LIN {X 0,Y 401.283,Z 772.145,A -85,B 0,C 180,E1 -11232.942,E2 -11232.942} C_VEL
LIN {X 0,Y 400.696,Z 783.943,A -85,B 0,C 180,E1 -11233.572,E2 -11233.572} C_VEL
LIN {X 0,Y 399.899,Z 796.285,A -85,B 0,C 180,E1 -11234.455,E2 -11234.455} C_VEL
LIN {X 0,Y 399.087,Z 807.279,A -85,B 0,C 180,E1 -11235.468,E2 -11235.468} C_VEL
LIN {X 0,Y 398.218,Z 818.113,A -85,B 0,C 180,E1 -11236.737,E2 -11236.737} C_VEL
LIN {X 0,Y 397.557,Z 826.911,A -85,B 0,C 180,E1 -11238.013,E2 -11238.013} C_VEL
LIN {X 0,Y 396.964,Z 834.155,A -85,B 0,C 180,E1 -11239.288,E2 -11239.288} C_VEL
LIN {X 0,Y 396.505,Z 841.253,A -85,B 0,C 180,E1 -11240.822,E2 -11240.822} C_VEL
LIN {X 0,Y 396.158,Z 846.888,A -85,B 0,C 180,E1 -11242.355,E2 -11242.355} C_VEL
LIN {X 0,Y 395.949,Z 851.307,A -85,B 0,C 180,E1 -11243.887,E2 -11243.887} C_VEL
LIN {X 0,Y 395.956,Z 853.636,A -85,B 0,C 180,E1 -11244.909,E2 -11244.909} C_VEL
LIN {X 0,Y 395.868,Z 855.53,A -85,B 0,C 180,E1 -11245.929,E2 -11245.929} C_VEL
LIN {X 0,Y 395.833,Z 856.959,A -85,B 0,C 180,E1 -11246.948,E2 -11246.948} C_VEL
LIN {X 0,Y 395.901,Z 857.969,A -85,B 0,C 180,E1 -11247.966,E2 -11247.966} C_VEL
LIN {X 0,Y 395.887,Z 858.585,A -85,B 0,C 180,E1 -11248.984,E2 -11248.984} C_VEL
LIN {X 0,Y 395.885,Z 858.804,A -85,B 0,C 180,E1 -11250.001,E2 -11250.001} C_VEL
LIN {X 0,Y 395.896,Z 857.963,A -85,B 0,C 180,E1 -11252.035,E2 -11252.035} C_VEL
LIN {X 0,Y 395.821,Z 856.95,A -85,B 0,C 180,E1 -11253.054,E2 -11253.054} C_VEL
LIN {X 0,Y 395.853,Z 855.516,A -85,B 0,C 180,E1 -11254.073,E2 -11254.073} C_VEL
LIN {X 0,Y 395.924,Z 852.533,A -85,B 0,C 180,E1 -11255.603,E2 -11255.603} C_VEL
LIN {X 0,Y 396.099,Z 848.483,A -85,B 0,C 180,E1 -11257.135,E2 -11257.135} C_VEL
LIN {X 0,Y 396.393,Z 842.229,A -85,B 0,C 180,E1 -11258.925,E2 -11258.925} C_VEL
LIN {X 0,Y 396.861,Z 835.406,A -85,B 0,C 180,E1 -11260.459,E2 -11260.459} C_VEL
LIN {X 0,Y 397.367,Z 828.432,A -85,B 0,C 180,E1 -11261.736,E2 -11261.736} C_VEL
LIN {X 0,Y 398.071,Z 820.005,A -85,B 0,C 180,E1 -11263.01,E2 -11263.01} C_VEL
LIN {X 0,Y 398.827,Z 809.551,A -85,B 0,C 180,E1 -11264.283,E2 -11264.283} C_VEL
LIN {X 0,Y 399.635,Z 799.186,A -85,B 0,C 180,E1 -11265.296,E2 -11265.296} C_VEL
LIN {X 0,Y 400.447,Z 787.762,A -85,B 0,C 180,E1 -11266.178,E2 -11266.178} C_VEL
LIN {X 0,Y 401.084,Z 775.888,A -85,B 0,C 180,E1 -11266.872,E2 -11266.872} C_VEL
LIN {X 0,Y 401.698,Z 763.05,A -85,B 0,C 180,E1 -11267.402,E2 -11267.402} C_VEL
LIN {X 0,Y 402.025,Z 751.019,A -85,B 0,C 180,E1 -11267.716,E2 -11267.716} C_VEL
LIN {X 0,Y 403.019,Z 672.877,A -85,B 0,C 180,E1 -11269.101,E2 -11269.101} C_VEL
LIN {X 0,Y 398.802,Z 636.907,A -85,B 0,C 180,E1 -11269.995,E2 -11269.995} C_VEL
LIN {X 0,Y 398.39,Z 632.093,A -85,B 0,C 180,E1 -11270.256,E2 -11270.256} C_VEL
LIN {X 0,Y 399.692,Z 611.54,A -85,B 0,C 180,E1 -11273.855,E2 -11273.855} C_VEL
LIN {X 0,Y 401.212,Z 590.111,A -85,B 0,C 180,E1 -11277.659,E2 -11277.659} C_VEL
LIN {X 0,Y 402.336,Z 576.283,A -85,B 0,C 180,E1 -11280.146,E2 -11280.146} C_VEL
LIN {X 0,Y 401.749,Z 571.846,A -85,B 0,C 180,E1 -11280.998,E2 -11280.998} C_VEL
LIN {X 0,Y 398.495,Z 556.913,A -85,B 0,C 180,E1 -11284.013,E2 -11284.013} C_VEL
LIN {X 0,Y 397.155,Z 551.015,A -85,B 0,C 180,E1 -11285.255,E2 -11285.255} C_VEL
LIN {X 0,Y 397.133,Z 551.019,A -85,B 0,C 180,E1 -11288.862,E2 -11288.862} C_VEL
LIN {X 0,Y 397.07,Z 551.022,A -85,B 0,C 180,E1 -11292.267,E2 -11292.267} C_VEL
LIN {X 0,Y 397.092,Z 551.018,A -85,B 0,C 180,E1 -11295.068,E2 -11295.068} C_VEL
LIN {X 0,Y 397.07,Z 551.014,A -85,B 0,C 180,E1 -11298.021,E2 -11298.021} C_VEL
LIN {X 0,Y 397.133,Z 551.019,A -85,B 0,C 180,E1 -11301.138,E2 -11301.138} C_VEL
LIN {X 0,Y 397.121,Z 551.01,A -85,B 0,C 180,E1 -11304.496,E2 -11304.496} C_VEL
LIN {X 0,Y 397.079,Z 551.013,A -85,B 0,C 180,E1 -11307.928,E2 -11307.928} C_VEL
LIN {X 0,Y 397.124,Z 551.02,A -85,B 0,C 180,E1 -11311.456,E2 -11311.456} C_VEL
LIN {X 0,Y 397.153,Z 551.003,A -85,B 0,C 180,E1 -11314.488,E2 -11314.488} C_VEL
LIN {X 0,Y 397.096,Z 551.018,A -85,B 0,C 180,E1 -11318.181,E2 -11318.181} C_VEL
LIN {X 0,Y 397.163,Z 550.999,A -85,B 0,C 180,E1 -11321.427,E2 -11321.427} C_VEL
LIN {X 0,Y 397.18,Z 551.005,A -85,B 0,C 180,E1 -11324.608,E2 -11324.608} C_VEL
LIN {X 0,Y 397.22,Z 550.997,A -85,B 0,C 180,E1 -11327.742,E2 -11327.742} C_VEL
LIN {X 0,Y 397.253,Z 550.988,A -85,B 0,C 180,E1 -11330.838,E2 -11330.838} C_VEL
LIN {X 0,Y 397.374,Z 550.985,A -85,B 0,C 180,E1 -11333.909,E2 -11333.909} C_VEL
LIN {X 0,Y 397.449,Z 550.962,A -85,B 0,C 180,E1 -11337.973,E2 -11337.973} C_VEL
LIN {X 0,Y 397.579,Z 550.961,A -85,B 0,C 180,E1 -11340,E2 -11340} C_VEL
LIN {X 0,Y 397.376,Z 550.981,A -85,B 0,C 180,E1 -11343.041,E2 -11343.041} C_VEL
LIN {X 0,Y 397.347,Z 550.978,A -85,B 0,C 180,E1 -11346.639,E2 -11346.639} C_VEL
LIN {X 0,Y 397.257,Z 550.999,A -85,B 0,C 180,E1 -11349.162,E2 -11349.162} C_VEL
LIN {X 0,Y 397.22,Z 550.989,A -85,B 0,C 180,E1 -11352.258,E2 -11352.258} C_VEL
LIN {X 0,Y 397.18,Z 551.008,A -85,B 0,C 180,E1 -11355.392,E2 -11355.392} C_VEL
LIN {X 0,Y 397.163,Z 550.998,A -85,B 0,C 180,E1 -11358.574,E2 -11358.574} C_VEL
LIN {X 0,Y 397.098,Z 551.02,A -85,B 0,C 180,E1 -11361.819,E2 -11361.819} C_VEL
LIN {X 0,Y 397.158,Z 551,A -85,B 0,C 180,E1 -11365.132,E2 -11365.132} C_VEL
LIN {X 0,Y 397.163,Z 551.012,A -85,B 0,C 180,E1 -11367.776,E2 -11367.776} C_VEL
LIN {X 0,Y 397.079,Z 551.013,A -85,B 0,C 180,E1 -11370.883,E2 -11370.883} C_VEL
LIN {X 0,Y 397.127,Z 551.013,A -85,B 0,C 180,E1 -11374.493,E2 -11374.493} C_VEL
LIN {X 0,Y 397.104,Z 551.022,A -85,B 0,C 180,E1 -11378.275,E2 -11378.275} C_VEL
LIN {X 0,Y 397.09,Z 551.022,A -85,B 0,C 180,E1 -11380.909,E2 -11380.909} C_VEL
LIN {X 0,Y 397.103,Z 551.014,A -85,B 0,C 180,E1 -11383.649,E2 -11383.649} C_VEL
LIN {X 0,Y 397.103,Z 551.006,A -85,B 0,C 180,E1 -11386.521,E2 -11386.521} C_VEL
LIN {X 0,Y 397.117,Z 551.018,A -85,B 0,C 180,E1 -11390.423,E2 -11390.423} C_VEL
LIN {X 0,Y 397.111,Z 551.021,A -85,B 0,C 180,E1 -11394.265,E2 -11394.265} C_VEL
LIN {X 0,Y 397.118,Z 551.023,A -85,B 0,C 180,E1 -11396.727,E2 -11396.727} C_VEL
LIN {X 0,Y 397.113,Z 551.129,A -85,B 0,C 180,E1 -11398.278,E2 -11398.278} C_VEL
LIN {X 0,Y 400.541,Z 564.762,A -85,B 0,C 180,E1 -11400.771,E2 -11400.771} C_VEL
LIN {X 0,Y 402.877,Z 576.265,A -85,B 0,C 180,E1 -11402.832,E2 -11402.832} C_VEL
LIN {X 0,Y 401.691,Z 596.601,A -85,B 0,C 180,E1 -11406.062,E2 -11406.062} C_VEL
LIN {X 0,Y 400.709,Z 617.149,A -85,B 0,C 180,E1 -11409.196,E2 -11409.196} C_VEL
LIN {X 0,Y 400.492,Z 622.956,A -85,B 0,C 180,E1 -11410.025,E2 -11410.025} C_VEL
LIN {X 0,Y 403.826,Z 644.421,A -85,B 0,C 180,E1 -11410.601,E2 -11410.601} C_VEL
LIN {X 0,Y 402.635,Z 734.616,A -85,B 0,C 180,E1 -11412.246,E2 -11412.246} C_VEL
LIN {X 0,Y 402.175,Z 747.681,A -85,B 0,C 180,E1 -11412.685,E2 -11412.685} C_VEL
LIN {X 0,Y 401.464,Z 760.645,A -85,B 0,C 180,E1 -11413.341,E2 -11413.341} C_VEL
LIN {X 0,Y 400.81,Z 771.721,A -85,B 0,C 180,E1 -11414.098,E2 -11414.098} C_VEL
LIN {X 0,Y 400.019,Z 782.969,A -85,B 0,C 180,E1 -11415.085,E2 -11415.085} C_VEL
LIN {X 0,Y 399.224,Z 793.487,A -85,B 0,C 180,E1 -11416.251,E2 -11416.251} C_VEL
LIN {X 0,Y 398.405,Z 802.783,A -85,B 0,C 180,E1 -11417.52,E2 -11417.52} C_VEL
LIN {X 0,Y 397.579,Z 811.736,A -85,B 0,C 180,E1 -11419.045,E2 -11419.045} C_VEL
LIN {X 0,Y 396.977,Z 818.928,A -85,B 0,C 180,E1 -11420.574,E2 -11420.574} C_VEL
LIN {X 0,Y 396.426,Z 825.533,A -85,B 0,C 180,E1 -11422.358,E2 -11422.358} C_VEL
LIN {X 0,Y 396.207,Z 829.864,A -85,B 0,C 180,E1 -11423.89,E2 -11423.89} C_VEL
LIN {X 0,Y 396.047,Z 832.144,A -85,B 0,C 180,E1 -11424.909,E2 -11424.909} C_VEL
LIN {X 0,Y 395.878,Z 834.005,A -85,B 0,C 180,E1 -11425.927,E2 -11425.927} C_VEL
LIN {X 0,Y 395.834,Z 836.097,A -85,B 0,C 180,E1 -11427.633,E2 -11427.633} C_VEL
LIN {X 0,Y 395.177,Z 836.822,A -85,B 0,C 180,E1 -11428.477,E2 -11428.477} C_VEL
LIN {X 0,Y 392.325,Z 837.458,A -85,B 0,C 180,E1 -11429.856,E2 -11429.856} C_VEL
LIN {X 0,Y 389.897,Z 837.369,A -85,B 0,C 180,E1 -11430.971,E2 -11430.971} C_VEL
LIN {X 0,Y 388.836,Z 836.891,A -85,B 0,C 180,E1 -11431.83,E2 -11431.83} C_VEL
LIN {X 0,Y 388.741,Z 836.644,A -85,B 0,C 180,E1 -11432.12,E2 -11432.12} C_VEL
LIN {X 0,Y 388.803,Z 834.362,A -85,B 0,C 180,E1 -11434.145,E2 -11434.145} C_VEL
LIN {X 0,Y 389.05,Z 831.49,A -85,B 0,C 180,E1 -11435.701,E2 -11435.701} C_VEL
LIN {X 0,Y 389.251,Z 827.592,A -85,B 0,C 180,E1 -11437.26,E2 -11437.26} C_VEL
LIN {X 0,Y 389.646,Z 822.542,A -85,B 0,C 180,E1 -11438.818,E2 -11438.818} C_VEL
LIN {X 0,Y 390.215,Z 816.176,A -85,B 0,C 180,E1 -11440.375,E2 -11440.375} C_VEL
LIN {X 0,Y 390.943,Z 808.254,A -85,B 0,C 180,E1 -11441.93,E2 -11441.93} C_VEL
LIN {X 0,Y 391.766,Z 800.152,A -85,B 0,C 180,E1 -11443.221,E2 -11443.221} C_VEL
LIN {X 0,Y 392.645,Z 790.211,A -85,B 0,C 180,E1 -11444.511,E2 -11444.511} C_VEL
LIN {X 0,Y 393.477,Z 779.041,A -85,B 0,C 180,E1 -11445.672,E2 -11445.672} C_VEL
LIN {X 0,Y 394.295,Z 768.089,A -85,B 0,C 180,E1 -11446.569,E2 -11446.569} C_VEL
LIN {X 0,Y 395.044,Z 755.761,A -85,B 0,C 180,E1 -11447.336,E2 -11447.336} C_VEL
LIN {X 0,Y 395.619,Z 742.937,A -85,B 0,C 180,E1 -11447.91,E2 -11447.91} C_VEL
LIN {X 0,Y 395.955,Z 730.774,A -85,B 0,C 180,E1 -11448.262,E2 -11448.262} C_VEL
LIN {X 0,Y 397.053,Z 646.296,A -85,B 0,C 180,E1 -11449.808,E2 -11449.808} C_VEL
LIN {X 0,Y 393.25,Z 623.873,A -85,B 0,C 180,E1 -11450.444,E2 -11450.444} C_VEL
LIN {X 0,Y 394.002,Z 604.702,A -85,B 0,C 180,E1 -11453.661,E2 -11453.661} C_VEL
LIN {X 0,Y 395.026,Z 588.085,A -85,B 0,C 180,E1 -11456.62,E2 -11456.62} C_VEL
LIN {X 0,Y 395.615,Z 576.878,A -85,B 0,C 180,E1 -11458.661,E2 -11458.661} C_VEL
LIN {X 0,Y 393.396,Z 565.484,A -85,B 0,C 180,E1 -11460.961,E2 -11460.961} C_VEL
LIN {X 0,Y 390.09,Z 551.892,A -85,B 0,C 180,E1 -11463.796,E2 -11463.796} C_VEL
LIN {X 0,Y 390.056,Z 551.895,A -85,B 0,C 180,E1 -11466.482,E2 -11466.482} C_VEL
LIN {X 0,Y 390.068,Z 551.89,A -85,B 0,C 180,E1 -11469.217,E2 -11469.217} C_VEL
LIN {X 0,Y 390.04,Z 551.896,A -85,B 0,C 180,E1 -11472.373,E2 -11472.373} C_VEL
LIN {X 0,Y 390.096,Z 551.892,A -85,B 0,C 180,E1 -11476.105,E2 -11476.105} C_VEL
LIN {X 0,Y 390.103,Z 551.892,A -85,B 0,C 180,E1 -11478.694,E2 -11478.694} C_VEL
LIN {X 0,Y 395.887,Z 568.43,A -85,B 0,C 180,E1 -11479.322,E2 -11479.322} C_VEL
LIN {X 0,Y 394.931,Z 631.63,A -85,B 0,C 180,E1 -11480.636,E2 -11480.636} C_VEL
LIN {X 0,Y 394.843,Z 645.21,A -85,B 0,C 180,E1 -11481.118,E2 -11481.118} C_VEL
LIN {X 0,Y 394.546,Z 657.641,A -85,B 0,C 180,E1 -11481.757,E2 -11481.757} C_VEL
LIN {X 0,Y 394.14,Z 668.866,A -85,B 0,C 180,E1 -11482.519,E2 -11482.519} C_VEL
LIN {X 0,Y 393.561,Z 680.822,A -85,B 0,C 180,E1 -11483.565,E2 -11483.565} C_VEL
LIN {X 0,Y 392.976,Z 691.857,A -85,B 0,C 180,E1 -11484.777,E2 -11484.777} C_VEL
LIN {X 0,Y 392.361,Z 700.866,A -85,B 0,C 180,E1 -11485.997,E2 -11485.997} C_VEL
LIN {X 0,Y 391.817,Z 709.636,A -85,B 0,C 180,E1 -11487.459,E2 -11487.459} C_VEL
LIN {X 0,Y 391.317,Z 716.667,A -85,B 0,C 180,E1 -11488.892,E2 -11488.892} C_VEL
LIN {X 0,Y 390.858,Z 722.55,A -85,B 0,C 180,E1 -11490.365,E2 -11490.365} C_VEL
LIN {X 0,Y 390.579,Z 728.004,A -85,B 0,C 180,E1 -11492.106,E2 -11492.106} C_VEL
LIN {X 0,Y 390.401,Z 730.789,A -85,B 0,C 180,E1 -11493.253,E2 -11493.253} C_VEL
LIN {X 0,Y 390.269,Z 733.041,A -85,B 0,C 180,E1 -11494.393,E2 -11494.393} C_VEL
LIN {X 0,Y 390.164,Z 734.702,A -85,B 0,C 180,E1 -11495.525,E2 -11495.525} C_VEL
LIN {X 0,Y 390.14,Z 735.967,A -85,B 0,C 180,E1 -11496.735,E2 -11496.735} C_VEL
LIN {X 0,Y 390.156,Z 736.561,A -85,B 0,C 180,E1 -11497.773,E2 -11497.773} C_VEL
LIN {X 0,Y 390.276,Z 736.668,A -85,B 0,C 180,E1 -11499.451,E2 -11499.451} C_VEL
LIN {X 0,Y 390.488,Z 735.718,A -85,B 0,C 180,E1 -11501.097,E2 -11501.097} C_VEL
LIN {X 0,Y 390.712,Z 734.208,A -85,B 0,C 180,E1 -11502.424,E2 -11502.424} C_VEL
LIN {X 0,Y 391.068,Z 731.78,A -85,B 0,C 180,E1 -11503.826,E2 -11503.826} C_VEL
LIN {X 0,Y 391.605,Z 727.154,A -85,B 0,C 180,E1 -11505.717,E2 -11505.717} C_VEL
LIN {X 0,Y 392.359,Z 720.839,A -85,B 0,C 180,E1 -11507.588,E2 -11507.588} C_VEL
LIN {X 0,Y 393.097,Z 713.912,A -85,B 0,C 180,E1 -11509.161,E2 -11509.161} C_VEL
LIN {X 0,Y 393.82,Z 706.604,A -85,B 0,C 180,E1 -11510.498,E2 -11510.498} C_VEL
LIN {X 0,Y 394.597,Z 697.843,A -85,B 0,C 180,E1 -11511.808,E2 -11511.808} C_VEL
LIN {X 0,Y 395.31,Z 688.161,A -85,B 0,C 180,E1 -11512.992,E2 -11512.992} C_VEL
LIN {X 0,Y 396.066,Z 677.186,A -85,B 0,C 180,E1 -11514.059,E2 -11514.059} C_VEL
LIN {X 0,Y 396.643,Z 666.019,A -85,B 0,C 180,E1 -11514.917,E2 -11514.917} C_VEL
LIN {X 0,Y 397.041,Z 654.125,A -85,B 0,C 180,E1 -11515.622,E2 -11515.622} C_VEL
LIN {X 0,Y 397.248,Z 640.901,A -85,B 0,C 180,E1 -11516.174,E2 -11516.174} C_VEL
LIN {X 0,Y 397.271,Z 622.782,A -85,B 0,C 180,E1 -11516.637,E2 -11516.637} C_VEL
LIN {X 0,Y 398.42,Z 570.844,A -85,B 0,C 180,E1 -11517.789,E2 -11517.789} C_VEL
LIN {X 0,Y 392.618,Z 557.28,A -85,B 0,C 180,E1 -11518.541,E2 -11518.541} C_VEL
LIN {X 0,Y 390.462,Z 552.491,A -85,B 0,C 180,E1 -11518.824,E2 -11518.824} C_VEL
LIN {X 0,Y 390.358,Z 551.864,A -85,B 0,C 180,E1 -11518.904,E2 -11518.904} C_VEL
LIN {X 0,Y 390.541,Z 551.84,A -85,B 0,C 180,E1 -11520,E2 -11520} C_VEL
LIN {X 0,Y 390.308,Z 551.867,A -85,B 0,C 180,E1 -11523.097,E2 -11523.097} C_VEL
LIN {X 0,Y 390.33,Z 551.864,A -85,B 0,C 180,E1 -11526.202,E2 -11526.202} C_VEL
LIN {X 0,Y 390.304,Z 551.865,A -85,B 0,C 180,E1 -11528.282,E2 -11528.282} C_VEL
LIN {X 0,Y 390.168,Z 551.881,A -85,B 0,C 180,E1 -11532.483,E2 -11532.483} C_VEL
LIN {X 0,Y 390.129,Z 551.881,A -85,B 0,C 180,E1 -11535.677,E2 -11535.677} C_VEL
LIN {X 0,Y 390.095,Z 551.895,A -85,B 0,C 180,E1 -11538.923,E2 -11538.923} C_VEL
LIN {X 0,Y 390.03,Z 551.901,A -85,B 0,C 180,E1 -11542.235,E2 -11542.235} C_VEL
LIN {X 0,Y 390.11,Z 551.889,A -85,B 0,C 180,E1 -11545.744,E2 -11545.744} C_VEL
LIN {X 0,Y 390.057,Z 551.898,A -85,B 0,C 180,E1 -11549.11,E2 -11549.11} C_VEL
LIN {X 0,Y 390.035,Z 551.902,A -85,B 0,C 180,E1 -11552.722,E2 -11552.722} C_VEL
LIN {X 0,Y 390.05,Z 551.898,A -85,B 0,C 180,E1 -11555.827,E2 -11555.827} C_VEL
LIN {X 0,Y 390.068,Z 551.897,A -85,B 0,C 180,E1 -11559.22,E2 -11559.22} C_VEL
LIN {X 0,Y 390.115,Z 551.891,A -85,B 0,C 180,E1 -11562.388,E2 -11562.388} C_VEL
LIN {X 0,Y 390.113,Z 551.891,A -85,B 0,C 180,E1 -11565.366,E2 -11565.366} C_VEL
LIN {X 0,Y 390.1,Z 551.894,A -85,B 0,C 180,E1 -11568.198,E2 -11568.198} C_VEL
LIN {X 0,Y 390.091,Z 551.895,A -85,B 0,C 180,E1 -11570.91,E2 -11570.91} C_VEL
LIN {X 0,Y 390.083,Z 551.899,A -85,B 0,C 180,E1 -11574.795,E2 -11574.795} C_VEL
LIN {X 0,Y 390.071,Z 551.916,A -85,B 0,C 180,E1 -11575.257,E2 -11575.257} C_VEL
LIN {X 0,Y 393.489,Z 565.056,A -85,B 0,C 180,E1 -11578.207,E2 -11578.207} C_VEL
LIN {X 0,Y 395.857,Z 576.032,A -85,B 0,C 180,E1 -11580.452,E2 -11580.452} C_VEL
LIN {X 0,Y 395.962,Z 579.686,A -85,B 0,C 180,E1 -11581.125,E2 -11581.125} C_VEL
LIN {X 0,Y 393.96,Z 600.394,A -85,B 0,C 180,E1 -11584.652,E2 -11584.652} C_VEL
LIN {X 0,Y 392.222,Z 623.137,A -85,B 0,C 180,E1 -11588.416,E2 -11588.416} C_VEL
LIN {X 0,Y 392.038,Z 625.864,A -85,B 0,C 180,E1 -11588.86,E2 -11588.86} C_VEL
LIN {X 0,Y 394.805,Z 646.803,A -85,B 0,C 180,E1 -11589.542,E2 -11589.542} C_VEL
LIN {X 0,Y 397.038,Z 672.475,A -85,B 0,C 180,E1 -11590.277,E2 -11590.277} C_VEL
LIN {X 0,Y 395.548,Z 739.472,A -85,B 0,C 180,E1 -11591.718,E2 -11591.718} C_VEL
LIN {X 0,Y 395.013,Z 761.303,A -85,B 0,C 180,E1 -11592.229,E2 -11592.229} C_VEL
LIN {X 0,Y 394.404,Z 774.608,A -85,B 0,C 180,E1 -11592.769,E2 -11592.769} C_VEL
LIN {X 0,Y 393.761,Z 785.751,A -85,B 0,C 180,E1 -11593.408,E2 -11593.408} C_VEL
LIN {X 0,Y 392.931,Z 797.671,A -85,B 0,C 180,E1 -11594.305,E2 -11594.305} C_VEL
LIN {X 0,Y 392.079,Z 808.27,A -85,B 0,C 180,E1 -11595.335,E2 -11595.335} C_VEL
LIN {X 0,Y 391.262,Z 817.929,A -85,B 0,C 180,E1 -11596.497,E2 -11596.497} C_VEL
LIN {X 0,Y 390.596,Z 826.726,A -85,B 0,C 180,E1 -11597.796,E2 -11597.796} C_VEL
LIN {X 0,Y 389.95,Z 833.967,A -85,B 0,C 180,E1 -11599.093,E2 -11599.093} C_VEL
LIN {X 0,Y 389.434,Z 841.062,A -85,B 0,C 180,E1 -11600.654,E2 -11600.654} C_VEL
LIN {X 0,Y 389.088,Z 846.697,A -85,B 0,C 180,E1 -11602.215,E2 -11602.215} C_VEL
LIN {X 0,Y 388.836,Z 851.863,A -85,B 0,C 180,E1 -11604.088,E2 -11604.088} C_VEL
LIN {X 0,Y 388.79,Z 855.338,A -85,B 0,C 180,E1 -11605.854,E2 -11605.854} C_VEL
LIN {X 0,Y 388.735,Z 856.767,A -85,B 0,C 180,E1 -11606.892,E2 -11606.892} C_VEL
LIN {X 0,Y 388.798,Z 857.776,A -85,B 0,C 180,E1 -11607.929,E2 -11607.929} C_VEL
LIN {X 0,Y 388.813,Z 858.393,A -85,B 0,C 180,E1 -11608.965,E2 -11608.965} C_VEL
LIN {X 0,Y 388.809,Z 858.612,A -85,B 0,C 180,E1 -11610.001,E2 -11610.001} C_VEL
LIN {X 0,Y 388.786,Z 858.388,A -85,B 0,C 180,E1 -11611.037,E2 -11611.037} C_VEL
LIN {X 0,Y 388.792,Z 857.77,A -85,B 0,C 180,E1 -11612.073,E2 -11612.073} C_VEL
LIN {X 0,Y 388.723,Z 856.757,A -85,B 0,C 180,E1 -11613.11,E2 -11613.11} C_VEL
LIN {X 0,Y 388.776,Z 855.323,A -85,B 0,C 180,E1 -11614.147,E2 -11614.147} C_VEL
LIN {X 0,Y 388.837,Z 851.846,A -85,B 0,C 180,E1 -11615.912,E2 -11615.912} C_VEL
LIN {X 0,Y 389.087,Z 846.672,A -85,B 0,C 180,E1 -11617.787,E2 -11617.787} C_VEL
LIN {X 0,Y 389.491,Z 839.928,A -85,B 0,C 180,E1 -11619.609,E2 -11619.609} C_VEL
LIN {X 0,Y 389.997,Z 832.563,A -85,B 0,C 180,E1 -11621.171,E2 -11621.171} C_VEL
LIN {X 0,Y 390.683,Z 825.051,A -85,B 0,C 180,E1 -11622.467,E2 -11622.467} C_VEL
LIN {X 0,Y 391.366,Z 816.46,A -85,B 0,C 180,E1 -11623.693,E2 -11623.693} C_VEL
LIN {X 0,Y 392.219,Z 805.746,A -85,B 0,C 180,E1 -11624.927,E2 -11624.927} C_VEL
LIN {X 0,Y 393.11,Z 794.436,A -85,B 0,C 180,E1 -11625.955,E2 -11625.955} C_VEL
LIN {X 0,Y 393.998,Z 782.649,A -85,B 0,C 180,E1 -11626.784,E2 -11626.784} C_VEL
LIN {X 0,Y 394.583,Z 770.308,A -85,B 0,C 180,E1 -11627.425,E2 -11627.425} C_VEL
LIN {X 0,Y 395.149,Z 756.569,A -85,B 0,C 180,E1 -11627.901,E2 -11627.901} C_VEL
LIN {X 0,Y 396.063,Z 693.26,A -85,B 0,C 180,E1 -11629.067,E2 -11629.067} C_VEL
LIN {X 0,Y 396.27,Z 673.243,A -85,B 0,C 180,E1 -11629.431,E2 -11629.431} C_VEL
LIN {X 0,Y 391.994,Z 637.185,A -85,B 0,C 180,E1 -11630.338,E2 -11630.338} C_VEL
LIN {X 0,Y 391.513,Z 630.548,A -85,B 0,C 180,E1 -11630.696,E2 -11630.696} C_VEL
LIN {X 0,Y 392.79,Z 610.387,A -85,B 0,C 180,E1 -11634.301,E2 -11634.301} C_VEL
LIN {X 0,Y 394.438,Z 588.982,A -85,B 0,C 180,E1 -11638.176,E2 -11638.176} C_VEL
LIN {X 0,Y 395.386,Z 576.632,A -85,B 0,C 180,E1 -11640.437,E2 -11640.437} C_VEL
LIN {X 0,Y 392.611,Z 563.044,A -85,B 0,C 180,E1 -11643.195,E2 -11643.195} C_VEL
LIN {X 0,Y 390.076,Z 551.897,A -85,B 0,C 180,E1 -11645.598,E2 -11645.598} C_VEL
LIN {X 0,Y 390.073,Z 551.898,A -85,B 0,C 180,E1 -11649.219,E2 -11649.219} C_VEL
LIN {X 0,Y 390.044,Z 551.898,A -85,B 0,C 180,E1 -11652.374,E2 -11652.374} C_VEL
LIN {X 0,Y 390.049,Z 551.899,A -85,B 0,C 180,E1 -11655.355,E2 -11655.355} C_VEL
LIN {X 0,Y 390.034,Z 551.89,A -85,B 0,C 180,E1 -11658.187,E2 -11658.187} C_VEL
LIN {X 0,Y 390.092,Z 551.894,A -85,B 0,C 180,E1 -11660.908,E2 -11660.908} C_VEL
LIN {X 0,Y 390.087,Z 551.888,A -85,B 0,C 180,E1 -11664.793,E2 -11664.793} C_VEL
LIN {X 0,Y 390.024,Z 551.891,A -85,B 0,C 180,E1 -11668.496,E2 -11668.496} C_VEL
LIN {X 0,Y 390.118,Z 551.888,A -85,B 0,C 180,E1 -11672.07,E2 -11672.07} C_VEL
LIN {X 0,Y 390.078,Z 551.882,A -85,B 0,C 180,E1 -11675.519,E2 -11675.519} C_VEL
LIN {X 0,Y 390.056,Z 551.897,A -85,B 0,C 180,E1 -11678.878,E2 -11678.878} C_VEL
LIN {X 0,Y 390.129,Z 551.87,A -85,B 0,C 180,E1 -11682.167,E2 -11682.167} C_VEL
LIN {X 0,Y 390.145,Z 551.887,A -85,B 0,C 180,E1 -11685.393,E2 -11685.393} C_VEL
LIN {X 0,Y 390.148,Z 551.873,A -85,B 0,C 180,E1 -11688.571,E2 -11688.571} C_VEL
LIN {X 0,Y 390.308,Z 551.865,A -85,B 0,C 180,E1 -11692.032,E2 -11692.032} C_VEL
LIN {X 0,Y 390.227,Z 551.872,A -85,B 0,C 180,E1 -11694.834,E2 -11694.834} C_VEL
LIN {X 0,Y 390.418,Z 551.837,A -85,B 0,C 180,E1 -11697.937,E2 -11697.937} C_VEL
LIN {X 0,Y 390.548,Z 551.837,A -85,B 0,C 180,E1 -11700,E2 -11700} C_VEL
LIN {X 0,Y 390.311,Z 551.861,A -85,B 0,C 180,E1 -11703.097,E2 -11703.097} C_VEL
LIN {X 0,Y 390.302,Z 551.856,A -85,B 0,C 180,E1 -11706.634,E2 -11706.634} C_VEL
LIN {X 0,Y 390.209,Z 551.878,A -85,B 0,C 180,E1 -11709.329,E2 -11709.329} C_VEL
LIN {X 0,Y 390.195,Z 551.866,A -85,B 0,C 180,E1 -11713.439,E2 -11713.439} C_VEL
LIN {X 0,Y 390.15,Z 551.883,A -85,B 0,C 180,E1 -11717.308,E2 -11717.308} C_VEL
LIN {X 0,Y 390.088,Z 551.889,A -85,B 0,C 180,E1 -11720.47,E2 -11720.47} C_VEL
LIN {X 0,Y 390.091,Z 551.892,A -85,B 0,C 180,E1 -11723.351,E2 -11723.351} C_VEL
LIN {X 0,Y 390.115,Z 551.886,A -85,B 0,C 180,E1 -11726.768,E2 -11726.768} C_VEL
LIN {X 0,Y 390.04,Z 551.891,A -85,B 0,C 180,E1 -11730.3,E2 -11730.3} C_VEL
LIN {X 0,Y 390.07,Z 551.898,A -85,B 0,C 180,E1 -11734.025,E2 -11734.025} C_VEL
LIN {X 0,Y 390.045,Z 551.9,A -85,B 0,C 180,E1 -11737.551,E2 -11737.551} C_VEL
LIN {X 0,Y 390.058,Z 551.898,A -85,B 0,C 180,E1 -11740.821,E2 -11740.821} C_VEL
LIN {X 0,Y 390.056,Z 551.893,A -85,B 0,C 180,E1 -11743.886,E2 -11743.886} C_VEL
LIN {X 0,Y 390.058,Z 551.881,A -85,B 0,C 180,E1 -11746.789,E2 -11746.789} C_VEL
LIN {X 0,Y 390.058,Z 551.897,A -85,B 0,C 180,E1 -11749.56,E2 -11749.56} C_VEL
LIN {X 0,Y 390.047,Z 551.89,A -85,B 0,C 180,E1 -11752.449,E2 -11752.449} C_VEL
LIN {X 0,Y 390.071,Z 551.898,A -85,B 0,C 180,E1 -11755.975,E2 -11755.975} C_VEL
LIN {X 0,Y 390.045,Z 551.911,A -85,B 0,C 180,E1 -11757.873,E2 -11757.873} C_VEL
LIN {X 0,Y 393.337,Z 564.739,A -85,B 0,C 180,E1 -11760.251,E2 -11760.251} C_VEL
LIN {X 0,Y 396.036,Z 577.286,A -85,B 0,C 180,E1 -11762.536,E2 -11762.536} C_VEL
LIN {X 0,Y 395.514,Z 587.469,A -85,B 0,C 180,E1 -11764.192,E2 -11764.192} C_VEL
LIN {X 0,Y 394.21,Z 610.213,A -85,B 0,C 180,E1 -11767.765,E2 -11767.765} C_VEL
LIN {X 0,Y 393.698,Z 623.087,A -85,B 0,C 180,E1 -11769.665,E2 -11769.665} C_VEL
LIN {X 0,Y 397.139,Z 644.951,A -85,B 0,C 180,E1 -11770.269,E2 -11770.269} C_VEL
LIN {X 0,Y 395.903,Z 734.743,A -85,B 0,C 180,E1 -11771.934,E2 -11771.934} C_VEL
LIN {X 0,Y 395.419,Z 747.843,A -85,B 0,C 180,E1 -11772.379,E2 -11772.379} C_VEL
LIN {X 0,Y 394.672,Z 760.818,A -85,B 0,C 180,E1 -11773.046,E2 -11773.046} C_VEL
LIN {X 0,Y 394.001,Z 771.9,A -85,B 0,C 180,E1 -11773.816,E2 -11773.816} C_VEL
LIN {X 0,Y 393.174,Z 783.072,A -85,B 0,C 180,E1 -11774.811,E2 -11774.811} C_VEL
LIN {X 0,Y 392.35,Z 793.674,A -85,B 0,C 180,E1 -11776.005,E2 -11776.005} C_VEL
LIN {X 0,Y 391.469,Z 802.973,A -85,B 0,C 180,E1 -11777.295,E2 -11777.295} C_VEL
LIN {X 0,Y 390.621,Z 811.927,A -85,B 0,C 180,E1 -11778.847,E2 -11778.847} C_VEL
LIN {X 0,Y 389.958,Z 819.12,A -85,B 0,C 180,E1 -11780.403,E2 -11780.403} C_VEL
LIN {X 0,Y 389.373,Z 825.726,A -85,B 0,C 180,E1 -11782.219,E2 -11782.219} C_VEL
LIN {X 0,Y 389.132,Z 830.057,A -85,B 0,C 180,E1 -11783.778,E2 -11783.778} C_VEL
LIN {X 0,Y 388.993,Z 832.337,A -85,B 0,C 180,E1 -11784.816,E2 -11784.816} C_VEL
LIN {X 0,Y 388.805,Z 834.198,A -85,B 0,C 180,E1 -11785.853,E2 -11785.853} C_VEL
LIN {X 0,Y 388.738,Z 836.329,A -85,B 0,C 180,E1 -11787.63,E2 -11787.63} C_VEL
LIN {X 0,Y 388.728,Z 837.229,A -85,B 0,C 180,E1 -11788.963,E2 -11788.963} C_VEL
LIN {X 0,Y 388.708,Z 837.465,A -85,B 0,C 180,E1 -11789.999,E2 -11789.999} C_VEL
LIN {X 0,Y 388.728,Z 837.274,A -85,B 0,C 180,E1 -11791.035,E2 -11791.035} C_VEL
LIN {X 0,Y 388.741,Z 836.644,A -85,B 0,C 180,E1 -11792.12,E2 -11792.12} C_VEL
LIN {X 0,Y 388.058,Z 835.905,A -85,B 0,C 180,E1 -11792.976,E2 -11792.976} C_VEL
LIN {X 0,Y 385.262,Z 834.163,A -85,B 0,C 180,E1 -11794.363,E2 -11794.363} C_VEL
LIN {X 0,Y 382.985,Z 832.294,A -85,B 0,C 180,E1 -11795.468,E2 -11795.468} C_VEL
LIN {X 0,Y 382.107,Z 830.538,A -85,B 0,C 180,E1 -11796.308,E2 -11796.308} C_VEL
LIN {X 0,Y 382.087,Z 829.881,A -85,B 0,C 180,E1 -11796.589,E2 -11796.589} C_VEL
LIN {X 0,Y 382.461,Z 824.529,A -85,B 0,C 180,E1 -11798.452,E2 -11798.452} C_VEL
LIN {X 0,Y 383.029,Z 818.635,A -85,B 0,C 180,E1 -11800.037,E2 -11800.037} C_VEL
LIN {X 0,Y 383.718,Z 811.296,A -85,B 0,C 180,E1 -11801.622,E2 -11801.622} C_VEL
LIN {X 0,Y 384.461,Z 803.784,A -85,B 0,C 180,E1 -11802.939,E2 -11802.939} C_VEL
LIN {X 0,Y 385.51,Z 793.585,A -85,B 0,C 180,E1 -11804.381,E2 -11804.381} C_VEL
LIN {X 0,Y 386.36,Z 782.728,A -85,B 0,C 180,E1 -11805.619,E2 -11805.619} C_VEL
LIN {X 0,Y 387.258,Z 771.636,A -85,B 0,C 180,E1 -11806.607,E2 -11806.607} C_VEL
LIN {X 0,Y 388.098,Z 759.358,A -85,B 0,C 180,E1 -11807.452,E2 -11807.452} C_VEL
LIN {X 0,Y 388.733,Z 746.404,A -85,B 0,C 180,E1 -11808.102,E2 -11808.102} C_VEL
LIN {X 0,Y 389.174,Z 733.502,A -85,B 0,C 180,E1 -11808.524,E2 -11808.524} C_VEL
LIN {X 0,Y 390.406,Z 647.315,A -85,B 0,C 180,E1 -11810.141,E2 -11810.141} C_VEL
LIN {X 0,Y 386.419,Z 623.901,A -85,B 0,C 180,E1 -11810.844,E2 -11810.844} C_VEL
LIN {X 0,Y 387.181,Z 606.286,A -85,B 0,C 180,E1 -11813.819,E2 -11813.819} C_VEL
LIN {X 0,Y 388.251,Z 589.054,A -85,B 0,C 180,E1 -11816.905,E2 -11816.905} C_VEL
LIN {X 0,Y 388.776,Z 578.115,A -85,B 0,C 180,E1 -11818.917,E2 -11818.917} C_VEL
LIN {X 0,Y 386.222,Z 565.725,A -85,B 0,C 180,E1 -11821.458,E2 -11821.458} C_VEL
LIN {X 0,Y 383.013,Z 552.776,A -85,B 0,C 180,E1 -11824.191,E2 -11824.191} C_VEL
LIN {X 0,Y 382.994,Z 552.782,A -85,B 0,C 180,E1 -11827.267,E2 -11827.267} C_VEL
LIN {X 0,Y 383.005,Z 552.77,A -85,B 0,C 180,E1 -11829.957,E2 -11829.957} C_VEL
LIN {X 0,Y 383,Z 552.766,A -85,B 0,C 180,E1 -11832.777,E2 -11832.777} C_VEL
LIN {X 0,Y 383.033,Z 552.773,A -85,B 0,C 180,E1 -11835.794,E2 -11835.794} C_VEL
LIN {X 0,Y 383.081,Z 552.767,A -85,B 0,C 180,E1 -11838.387,E2 -11838.387} C_VEL
LIN {X 0,Y 389.013,Z 569.772,A -85,B 0,C 180,E1 -11839.055,E2 -11839.055} C_VEL
LIN {X 0,Y 388.083,Z 632.568,A -85,B 0,C 180,E1 -11840.393,E2 -11840.393} C_VEL
LIN {X 0,Y 387.971,Z 646.052,A -85,B 0,C 180,E1 -11840.88,E2 -11840.88} C_VEL
LIN {X 0,Y 387.656,Z 658.819,A -85,B 0,C 180,E1 -11841.549,E2 -11841.549} C_VEL
LIN {X 0,Y 387.181,Z 671.323,A -85,B 0,C 180,E1 -11842.434,E2 -11842.434} C_VEL
LIN {X 0,Y 386.625,Z 682.659,A -85,B 0,C 180,E1 -11843.464,E2 -11843.464} C_VEL
LIN {X 0,Y 386.051,Z 692.741,A -85,B 0,C 180,E1 -11844.598,E2 -11844.598} C_VEL
LIN {X 0,Y 385.394,Z 702.11,A -85,B 0,C 180,E1 -11845.892,E2 -11845.892} C_VEL
LIN {X 0,Y 384.78,Z 711.29,A -85,B 0,C 180,E1 -11847.461,E2 -11847.461} C_VEL
LIN {X 0,Y 384.291,Z 718.091,A -85,B 0,C 180,E1 -11848.892,E2 -11848.892} C_VEL
LIN {X 0,Y 383.824,Z 723.831,A -85,B 0,C 180,E1 -11850.371,E2 -11850.371} C_VEL
LIN {X 0,Y 383.555,Z 729.21,A -85,B 0,C 180,E1 -11852.144,E2 -11852.144} C_VEL
LIN {X 0,Y 383.29,Z 733.253,A -85,B 0,C 180,E1 -11853.953,E2 -11853.953} C_VEL
LIN {X 0,Y 383.184,Z 735.08,A -85,B 0,C 180,E1 -11855.049,E2 -11855.049} C_VEL
LIN {X 0,Y 383.106,Z 736.769,A -85,B 0,C 180,E1 -11856.522,E2 -11856.522} C_VEL
LIN {X 0,Y 383.173,Z 737.797,A -85,B 0,C 180,E1 -11858.48,E2 -11858.48} C_VEL
LIN {X 0,Y 383.278,Z 737.701,A -85,B 0,C 180,E1 -11859.611,E2 -11859.611} C_VEL
LIN {X 0,Y 383.434,Z 737.167,A -85,B 0,C 180,E1 -11860.736,E2 -11860.736} C_VEL
LIN {X 0,Y 383.671,Z 735.655,A -85,B 0,C 180,E1 -11862.268,E2 -11862.268} C_VEL
LIN {X 0,Y 384.145,Z 732.706,A -85,B 0,C 180,E1 -11864.072,E2 -11864.072} C_VEL
LIN {X 0,Y 384.598,Z 729.182,A -85,B 0,C 180,E1 -11865.574,E2 -11865.574} C_VEL
LIN {X 0,Y 385.307,Z 723.609,A -85,B 0,C 180,E1 -11867.357,E2 -11867.357} C_VEL
LIN {X 0,Y 386.116,Z 716.774,A -85,B 0,C 180,E1 -11869.035,E2 -11869.035} C_VEL
LIN {X 0,Y 386.981,Z 708.801,A -85,B 0,C 180,E1 -11870.593,E2 -11870.593} C_VEL
LIN {X 0,Y 387.772,Z 700.306,A -85,B 0,C 180,E1 -11871.925,E2 -11871.925} C_VEL
LIN {X 0,Y 388.556,Z 690.663,A -85,B 0,C 180,E1 -11873.157,E2 -11873.157} C_VEL
LIN {X 0,Y 389.362,Z 679.833,A -85,B 0,C 180,E1 -11874.268,E2 -11874.268} C_VEL
LIN {X 0,Y 390.037,Z 667.89,A -85,B 0,C 180,E1 -11875.22,E2 -11875.22} C_VEL
LIN {X 0,Y 390.509,Z 654.994,A -85,B 0,C 180,E1 -11876.001,E2 -11876.001} C_VEL
LIN {X 0,Y 390.731,Z 641.923,A -85,B 0,C 180,E1 -11876.552,E2 -11876.552} C_VEL
LIN {X 0,Y 390.772,Z 623.164,A -85,B 0,C 180,E1 -11877.043,E2 -11877.043} C_VEL
LIN {X 0,Y 392.006,Z 572.731,A -85,B 0,C 180,E1 -11878.192,E2 -11878.192} C_VEL
LIN {X 0,Y 386.596,Z 560.133,A -85,B 0,C 180,E1 -11878.92,E2 -11878.92} C_VEL
LIN {X 0,Y 383.49,Z 553.413,A -85,B 0,C 180,E1 -11879.344,E2 -11879.344} C_VEL
LIN {X 0,Y 383.375,Z 552.734,A -85,B 0,C 180,E1 -11879.409,E2 -11879.409} C_VEL
LIN {X 0,Y 383.314,Z 552.741,A -85,B 0,C 180,E1 -11881.051,E2 -11881.051} C_VEL
LIN {X 0,Y 383.245,Z 552.747,A -85,B 0,C 180,E1 -11883.154,E2 -11883.154} C_VEL
LIN {X 0,Y 383.286,Z 552.742,A -85,B 0,C 180,E1 -11886.316,E2 -11886.316} C_VEL
LIN {X 0,Y 383.25,Z 552.745,A -85,B 0,C 180,E1 -11888.436,E2 -11888.436} C_VEL
LIN {X 0,Y 383.097,Z 552.764,A -85,B 0,C 180,E1 -11891.642,E2 -11891.642} C_VEL
LIN {X 0,Y 383.102,Z 552.762,A -85,B 0,C 180,E1 -11894.882,E2 -11894.882} C_VEL
LIN {X 0,Y 383.079,Z 552.766,A -85,B 0,C 180,E1 -11898.173,E2 -11898.173} C_VEL
LIN {X 0,Y 382.983,Z 552.778,A -85,B 0,C 180,E1 -11901.532,E2 -11901.532} C_VEL
LIN {X 0,Y 383.043,Z 552.773,A -85,B 0,C 180,E1 -11904.961,E2 -11904.961} C_VEL
LIN {X 0,Y 383.04,Z 552.772,A -85,B 0,C 180,E1 -11908.493,E2 -11908.493} C_VEL
LIN {X 0,Y 383.003,Z 552.776,A -85,B 0,C 180,E1 -11912.15,E2 -11912.15} C_VEL
LIN {X 0,Y 383.01,Z 552.771,A -85,B 0,C 180,E1 -11914.669,E2 -11914.669} C_VEL
LIN {X 0,Y 382.996,Z 552.773,A -85,B 0,C 180,E1 -11917.906,E2 -11917.906} C_VEL
LIN {X 0,Y 383.04,Z 552.775,A -85,B 0,C 180,E1 -11921.34,E2 -11921.34} C_VEL
LIN {X 0,Y 383.063,Z 552.772,A -85,B 0,C 180,E1 -11924.316,E2 -11924.316} C_VEL
LIN {X 0,Y 383.069,Z 552.768,A -85,B 0,C 180,E1 -11927.25,E2 -11927.25} C_VEL
LIN {X 0,Y 383.018,Z 552.775,A -85,B 0,C 180,E1 -11930.413,E2 -11930.413} C_VEL
LIN {X 0,Y 383.023,Z 552.779,A -85,B 0,C 180,E1 -11934.046,E2 -11934.046} C_VEL
LIN {X 0,Y 383.055,Z 552.933,A -85,B 0,C 180,E1 -11934.736,E2 -11934.736} C_VEL
LIN {X 0,Y 385.913,Z 563.614,A -85,B 0,C 180,E1 -11937.254,E2 -11937.254} C_VEL
LIN {X 0,Y 388.69,Z 575.718,A -85,B 0,C 180,E1 -11939.853,E2 -11939.853} C_VEL
LIN {X 0,Y 389.285,Z 579.464,A -85,B 0,C 180,E1 -11940.607,E2 -11940.607} C_VEL
LIN {X 0,Y 387.538,Z 596.64,A -85,B 0,C 180,E1 -11943.622,E2 -11943.622} C_VEL
LIN {X 0,Y 385.709,Z 617.795,A -85,B 0,C 180,E1 -11947.221,E2 -11947.221} C_VEL
LIN {X 0,Y 385.222,Z 624.537,A -85,B 0,C 180,E1 -11948.355,E2 -11948.355} C_VEL
LIN {X 0,Y 388.031,Z 645.109,A -85,B 0,C 180,E1 -11949.064,E2 -11949.064} C_VEL
LIN {X 0,Y 390.138,Z 668.772,A -85,B 0,C 180,E1 -11949.763,E2 -11949.763} C_VEL
LIN {X 0,Y 390.407,Z 676.656,A -85,B 0,C 180,E1 -11949.966,E2 -11949.966} C_VEL
LIN {X 0,Y 388.901,Z 738.029,A -85,B 0,C 180,E1 -11951.326,E2 -11951.326} C_VEL
LIN {X 0,Y 388.645,Z 747.872,A -85,B 0,C 180,E1 -11951.586,E2 -11951.586} C_VEL
LIN {X 0,Y 388.277,Z 761.184,A -85,B 0,C 180,E1 -11951.91,E2 -11951.91} C_VEL
LIN {X 0,Y 387.613,Z 774.457,A -85,B 0,C 180,E1 -11952.457,E2 -11952.457} C_VEL
LIN {X 0,Y 386.807,Z 787.544,A -85,B 0,C 180,E1 -11953.237,E2 -11953.237} C_VEL
LIN {X 0,Y 385.952,Z 798.924,A -85,B 0,C 180,E1 -11954.15,E2 -11954.15} C_VEL
LIN {X 0,Y 385.095,Z 809.257,A -85,B 0,C 180,E1 -11955.198,E2 -11955.198} C_VEL
LIN {X 0,Y 384.211,Z 819.684,A -85,B 0,C 180,E1 -11956.514,E2 -11956.514} C_VEL
LIN {X 0,Y 383.483,Z 828.104,A -85,B 0,C 180,E1 -11957.834,E2 -11957.834} C_VEL
LIN {X 0,Y 382.746,Z 836.303,A -85,B 0,C 180,E1 -11959.42,E2 -11959.42} C_VEL
LIN {X 0,Y 382.283,Z 842.891,A -85,B 0,C 180,E1 -11961.011,E2 -11961.011} C_VEL
LIN {X 0,Y 381.946,Z 848.122,A -85,B 0,C 180,E1 -11962.601,E2 -11962.601} C_VEL
LIN {X 0,Y 381.737,Z 852.045,A -85,B 0,C 180,E1 -11964.137,E2 -11964.137} C_VEL
LIN {X 0,Y 381.714,Z 855.146,A -85,B 0,C 180,E1 -11965.777,E2 -11965.777} C_VEL
LIN {X 0,Y 381.642,Z 856.574,A -85,B 0,C 180,E1 -11966.834,E2 -11966.834} C_VEL
LIN {X 0,Y 381.694,Z 857.583,A -85,B 0,C 180,E1 -11967.891,E2 -11967.891} C_VEL
LIN {X 0,Y 381.741,Z 858.201,A -85,B 0,C 180,E1 -11968.946,E2 -11968.946} C_VEL
LIN {X 0,Y 381.735,Z 858.42,A -85,B 0,C 180,E1 -11970.001,E2 -11970.001} C_VEL
LIN {X 0,Y 381.716,Z 858.196,A -85,B 0,C 180,E1 -11971.056,E2 -11971.056} C_VEL
LIN {X 0,Y 381.688,Z 857.576,A -85,B 0,C 180,E1 -11972.111,E2 -11972.111} C_VEL
LIN {X 0,Y 381.63,Z 856.564,A -85,B 0,C 180,E1 -11973.168,E2 -11973.168} C_VEL
LIN {X 0,Y 381.701,Z 855.13,A -85,B 0,C 180,E1 -11974.224,E2 -11974.224} C_VEL
LIN {X 0,Y 381.737,Z 852.03,A -85,B 0,C 180,E1 -11975.862,E2 -11975.862} C_VEL
LIN {X 0,Y 381.958,Z 848.097,A -85,B 0,C 180,E1 -11977.401,E2 -11977.401} C_VEL
LIN {X 0,Y 382.296,Z 841.843,A -85,B 0,C 180,E1 -11979.257,E2 -11979.257} C_VEL
LIN {X 0,Y 382.795,Z 835.022,A -85,B 0,C 180,E1 -11980.848,E2 -11980.848} C_VEL
LIN {X 0,Y 383.443,Z 828.052,A -85,B 0,C 180,E1 -11982.169,E2 -11982.169} C_VEL
LIN {X 0,Y 384.18,Z 819.628,A -85,B 0,C 180,E1 -11983.489,E2 -11983.489} C_VEL
LIN {X 0,Y 385.043,Z 809.18,A -85,B 0,C 180,E1 -11984.806,E2 -11984.806} C_VEL
LIN {X 0,Y 385.922,Z 798.823,A -85,B 0,C 180,E1 -11985.853,E2 -11985.853} C_VEL
LIN {X 0,Y 386.808,Z 787.411,A -85,B 0,C 180,E1 -11986.765,E2 -11986.765} C_VEL
LIN {X 0,Y 387.495,Z 775.556,A -85,B 0,C 180,E1 -11987.482,E2 -11987.482} C_VEL
LIN {X 0,Y 388.177,Z 762.754,A -85,B 0,C 180,E1 -11988.029,E2 -11988.029} C_VEL
LIN {X 0,Y 388.557,Z 750.806,A -85,B 0,C 180,E1 -11988.351,E2 -11988.351} C_VEL
LIN {X 0,Y 389.553,Z 673.809,A -85,B 0,C 180,E1 -11989.768,E2 -11989.768} C_VEL
LIN {X 0,Y 385.462,Z 638.824,A -85,B 0,C 180,E1 -11990.662,E2 -11990.662} C_VEL
LIN {X 0,Y 384.993,Z 634.332,A -85,B 0,C 180,E1 -11990.863,E2 -11990.863} C_VEL
LIN {X 0,Y 384.587,Z 628.881,A -85,B 0,C 180,E1 -11991.172,E2 -11991.172} C_VEL
LIN {X 0,Y 385.923,Z 609.198,A -85,B 0,C 180,E1 -11994.763,E2 -11994.763} C_VEL
LIN {X 0,Y 387.657,Z 587.77,A -85,B 0,C 180,E1 -11998.714,E2 -11998.714} C_VEL
LIN {X 0,Y 388.457,Z 578.542,A -85,B 0,C 180,E1 -12000.437,E2 -12000.437} C_VEL
LIN {X 0,Y 386.641,Z 568.814,A -85,B 0,C 180,E1 -12002.427,E2 -12002.427} C_VEL
LIN {X 0,Y 383.292,Z 553.909,A -85,B 0,C 180,E1 -12005.603,E2 -12005.603} C_VEL
LIN {X 0,Y 383.012,Z 552.776,A -85,B 0,C 180,E1 -12005.876,E2 -12005.876} C_VEL
LIN {X 0,Y 383.018,Z 552.775,A -85,B 0,C 180,E1 -12009.587,E2 -12009.587} C_VEL
LIN {X 0,Y 383.007,Z 552.778,A -85,B 0,C 180,E1 -12012.779,E2 -12012.779} C_VEL
LIN {X 0,Y 383.002,Z 552.776,A -85,B 0,C 180,E1 -12015.79,E2 -12015.79} C_VEL
LIN {X 0,Y 382.99,Z 552.768,A -85,B 0,C 180,E1 -12018.796,E2 -12018.796} C_VEL
LIN {X 0,Y 383.002,Z 552.771,A -85,B 0,C 180,E1 -12022.096,E2 -12022.096} C_VEL
LIN {X 0,Y 383.02,Z 552.775,A -85,B 0,C 180,E1 -12025.332,E2 -12025.332} C_VEL
LIN {X 0,Y 382.984,Z 552.766,A -85,B 0,C 180,E1 -12029.081,E2 -12029.081} C_VEL
LIN {X 0,Y 383.058,Z 552.768,A -85,B 0,C 180,E1 -12032.698,E2 -12032.698} C_VEL
LIN {X 0,Y 383.051,Z 552.757,A -85,B 0,C 180,E1 -12035.04,E2 -12035.04} C_VEL
LIN {X 0,Y 382.993,Z 552.775,A -85,B 0,C 180,E1 -12038.469,E2 -12038.469} C_VEL
LIN {X 0,Y 383.064,Z 552.75,A -85,B 0,C 180,E1 -12041.826,E2 -12041.826} C_VEL
LIN {X 0,Y 383.111,Z 552.76,A -85,B 0,C 180,E1 -12045.118,E2 -12045.118} C_VEL
LIN {X 0,Y 383.097,Z 552.751,A -85,B 0,C 180,E1 -12048.358,E2 -12048.358} C_VEL
LIN {X 0,Y 383.264,Z 552.743,A -85,B 0,C 180,E1 -12051.976,E2 -12051.976} C_VEL
LIN {X 0,Y 383.199,Z 552.747,A -85,B 0,C 180,E1 -12054.739,E2 -12054.739} C_VEL
LIN {X 0,Y 383.385,Z 552.712,A -85,B 0,C 180,E1 -12057.899,E2 -12057.899} C_VEL
LIN {X 0,Y 383.518,Z 552.713,A -85,B 0,C 180,E1 -12060,E2 -12060} C_VEL
LIN {X 0,Y 383.248,Z 552.741,A -85,B 0,C 180,E1 -12063.154,E2 -12063.154} C_VEL
LIN {X 0,Y 383.262,Z 552.734,A -85,B 0,C 180,E1 -12066.626,E2 -12066.626} C_VEL
LIN {X 0,Y 383.155,Z 552.758,A -85,B 0,C 180,E1 -12069.502,E2 -12069.502} C_VEL
LIN {X 0,Y 383.126,Z 552.747,A -85,B 0,C 180,E1 -12073.536,E2 -12073.536} C_VEL
LIN {X 0,Y 383.096,Z 552.763,A -85,B 0,C 180,E1 -12077.455,E2 -12077.455} C_VEL
LIN {X 0,Y 383.03,Z 552.768,A -85,B 0,C 180,E1 -12080.647,E2 -12080.647} C_VEL
LIN {X 0,Y 383.034,Z 552.769,A -85,B 0,C 180,E1 -12083.807,E2 -12083.807} C_VEL
LIN {X 0,Y 383.081,Z 552.757,A -85,B 0,C 180,E1 -12086.123,E2 -12086.123} C_VEL
LIN {X 0,Y 382.993,Z 552.775,A -85,B 0,C 180,E1 -12089.7,E2 -12089.7} C_VEL
LIN {X 0,Y 383.005,Z 552.776,A -85,B 0,C 180,E1 -12093.401,E2 -12093.401} C_VEL
LIN {X 0,Y 383.033,Z 552.769,A -85,B 0,C 180,E1 -12096.165,E2 -12096.165} C_VEL
LIN {X 0,Y 383.01,Z 552.772,A -85,B 0,C 180,E1 -12099.958,E2 -12099.958} C_VEL
LIN {X 0,Y 383.007,Z 552.77,A -85,B 0,C 180,E1 -12102.779,E2 -12102.779} C_VEL
LIN {X 0,Y 382.999,Z 552.774,A -85,B 0,C 180,E1 -12105.789,E2 -12105.789} C_VEL
LIN {X 0,Y 382.989,Z 552.772,A -85,B 0,C 180,E1 -12108.796,E2 -12108.796} C_VEL
LIN {X 0,Y 383.003,Z 552.765,A -85,B 0,C 180,E1 -12112.096,E2 -12112.096} C_VEL
LIN {X 0,Y 383.021,Z 552.776,A -85,B 0,C 180,E1 -12115.332,E2 -12115.332} C_VEL
LIN {X 0,Y 383.034,Z 552.955,A -85,B 0,C 180,E1 -12117.474,E2 -12117.474} C_VEL
LIN {X 0,Y 386.479,Z 566.231,A -85,B 0,C 180,E1 -12119.995,E2 -12119.995} C_VEL
LIN {X 0,Y 389.131,Z 578.45,A -85,B 0,C 180,E1 -12122.249,E2 -12122.249} C_VEL
LIN {X 0,Y 389.175,Z 582.468,A -85,B 0,C 180,E1 -12122.931,E2 -12122.931} C_VEL
LIN {X 0,Y 387.809,Z 603.008,A -85,B 0,C 180,E1 -12126.22,E2 -12126.22} C_VEL
LIN {X 0,Y 387.018,Z 621.241,A -85,B 0,C 180,E1 -12129.01,E2 -12129.01} C_VEL
LIN {X 0,Y 386.989,Z 623.532,A -85,B 0,C 180,E1 -12129.308,E2 -12129.308} C_VEL
LIN {X 0,Y 390.474,Z 645.902,A -85,B 0,C 180,E1 -12129.934,E2 -12129.934} C_VEL
LIN {X 0,Y 389.169,Z 734.871,A -85,B 0,C 180,E1 -12131.61,E2 -12131.61} C_VEL
LIN {X 0,Y 388.67,Z 748.004,A -85,B 0,C 180,E1 -12132.063,E2 -12132.063} C_VEL
LIN {X 0,Y 387.893,Z 760.991,A -85,B 0,C 180,E1 -12132.741,E2 -12132.741} C_VEL
LIN {X 0,Y 387.208,Z 772.08,A -85,B 0,C 180,E1 -12133.524,E2 -12133.524} C_VEL
LIN {X 0,Y 386.409,Z 782.183,A -85,B 0,C 180,E1 -12134.425,E2 -12134.425} C_VEL
LIN {X 0,Y 385.58,Z 792.826,A -85,B 0,C 180,E1 -12135.62,E2 -12135.62} C_VEL
LIN {X 0,Y 384.547,Z 803.162,A -85,B 0,C 180,E1 -12137.062,E2 -12137.062} C_VEL
LIN {X 0,Y 383.797,Z 810.785,A -85,B 0,C 180,E1 -12138.379,E2 -12138.379} C_VEL
LIN {X 0,Y 383.08,Z 818.223,A -85,B 0,C 180,E1 -12139.962,E2 -12139.962} C_VEL
LIN {X 0,Y 382.471,Z 824.198,A -85,B 0,C 180,E1 -12141.546,E2 -12141.546} C_VEL
LIN {X 0,Y 382.16,Z 829.232,A -85,B 0,C 180,E1 -12143.254,E2 -12143.254} C_VEL
LIN {X 0,Y 381.918,Z 832.53,A -85,B 0,C 180,E1 -12144.72,E2 -12144.72} C_VEL
LIN {X 0,Y 381.736,Z 834.391,A -85,B 0,C 180,E1 -12145.776,E2 -12145.776} C_VEL
LIN {X 0,Y 381.667,Z 835.813,A -85,B 0,C 180,E1 -12146.832,E2 -12146.832} C_VEL
LIN {X 0,Y 381.643,Z 837.422,A -85,B 0,C 180,E1 -12148.944,E2 -12148.944} C_VEL
LIN {X 0,Y 381.64,Z 837.657,A -85,B 0,C 180,E1 -12149.999,E2 -12149.999} C_VEL
LIN {X 0,Y 381.643,Z 837.466,A -85,B 0,C 180,E1 -12151.054,E2 -12151.054} C_VEL
LIN {X 0,Y 381.655,Z 835.917,A -85,B 0,C 180,E1 -12153.166,E2 -12153.166} C_VEL
LIN {X 0,Y 381.734,Z 834.553,A -85,B 0,C 180,E1 -12154.222,E2 -12154.222} C_VEL
LIN {X 0,Y 381.986,Z 831.681,A -85,B 0,C 180,E1 -12155.807,E2 -12155.807} C_VEL
LIN {X 0,Y 382.087,Z 829.881,A -85,B 0,C 180,E1 -12156.589,E2 -12156.589} C_VEL
LIN {X 0,Y 381.613,Z 827.821,A -85,B 0,C 180,E1 -12157.416,E2 -12157.416} C_VEL
LIN {X 0,Y 379.084,Z 824.033,A -85,B 0,C 180,E1 -12158.744,E2 -12158.744} C_VEL
LIN {X 0,Y 376.611,Z 819.552,A -85,B 0,C 180,E1 -12160.037,E2 -12160.037} C_VEL
LIN {X 0,Y 376.233,Z 816.403,A -85,B 0,C 180,E1 -12160.799,E2 -12160.799} C_VEL
LIN {X 0,Y 377.026,Z 808.625,A -85,B 0,C 180,E1 -12162.377,E2 -12162.377} C_VEL
LIN {X 0,Y 377.979,Z 800.517,A -85,B 0,C 180,E1 -12163.712,E2 -12163.712} C_VEL
LIN {X 0,Y 378.885,Z 790.568,A -85,B 0,C 180,E1 -12165.05,E2 -12165.05} C_VEL
LIN {X 0,Y 379.835,Z 779.388,A -85,B 0,C 180,E1 -12166.25,E2 -12166.25} C_VEL
LIN {X 0,Y 380.717,Z 768.42,A -85,B 0,C 180,E1 -12167.178,E2 -12167.178} C_VEL
LIN {X 0,Y 381.554,Z 756.063,A -85,B 0,C 180,E1 -12167.969,E2 -12167.969} C_VEL
LIN {X 0,Y 382.15,Z 743.196,A -85,B 0,C 180,E1 -12168.564,E2 -12168.564} C_VEL
LIN {X 0,Y 382.53,Z 730.904,A -85,B 0,C 180,E1 -12168.927,E2 -12168.927} C_VEL
LIN {X 0,Y 383.743,Z 648.063,A -85,B 0,C 180,E1 -12170.492,E2 -12170.492} C_VEL
LIN {X 0,Y 379.591,Z 624.027,A -85,B 0,C 180,E1 -12171.234,E2 -12171.234} C_VEL
LIN {X 0,Y 380.415,Z 606.241,A -85,B 0,C 180,E1 -12174.27,E2 -12174.27} C_VEL
LIN {X 0,Y 381.564,Z 588.872,A -85,B 0,C 180,E1 -12177.416,E2 -12177.416} C_VEL
LIN {X 0,Y 382.039,Z 580.983,A -85,B 0,C 180,E1 -12178.873,E2 -12178.873} C_VEL
LIN {X 0,Y 380.619,Z 572.988,A -85,B 0,C 180,E1 -12180.514,E2 -12180.514} C_VEL
LIN {X 0,Y 377.751,Z 560.498,A -85,B 0,C 180,E1 -12183.152,E2 -12183.152} C_VEL
LIN {X 0,Y 375.973,Z 553.657,A -85,B 0,C 180,E1 -12184.62,E2 -12184.62} C_VEL
LIN {X 0,Y 375.972,Z 553.655,A -85,B 0,C 180,E1 -12188.27,E2 -12188.27} C_VEL
LIN {X 0,Y 375.931,Z 553.658,A -85,B 0,C 180,E1 -12191.6,E2 -12191.6} C_VEL
LIN {X 0,Y 375.974,Z 553.648,A -85,B 0,C 180,E1 -12195.259,E2 -12195.259} C_VEL
LIN {X 0,Y 376.046,Z 553.643,A -85,B 0,C 180,E1 -12198.093,E2 -12198.093} C_VEL
LIN {X 0,Y 382.222,Z 571.275,A -85,B 0,C 180,E1 -12198.794,E2 -12198.794} C_VEL
LIN {X 0,Y 381.211,Z 633.153,A -85,B 0,C 180,E1 -12200.143,E2 -12200.143} C_VEL
LIN {X 0,Y 381.093,Z 646.485,A -85,B 0,C 180,E1 -12200.627,E2 -12200.627} C_VEL
LIN {X 0,Y 380.785,Z 659.263,A -85,B 0,C 180,E1 -12201.302,E2 -12201.302} C_VEL
LIN {X 0,Y 380.344,Z 670.561,A -85,B 0,C 180,E1 -12202.092,E2 -12202.092} C_VEL
LIN {X 0,Y 379.723,Z 682.788,A -85,B 0,C 180,E1 -12203.197,E2 -12203.197} C_VEL
LIN {X 0,Y 379.104,Z 693.482,A -85,B 0,C 180,E1 -12204.408,E2 -12204.408} C_VEL
LIN {X 0,Y 378.406,Z 703.487,A -85,B 0,C 180,E1 -12205.818,E2 -12205.818} C_VEL
LIN {X 0,Y 377.783,Z 712.275,A -85,B 0,C 180,E1 -12207.35,E2 -12207.35} C_VEL
LIN {X 0,Y 377.245,Z 719.804,A -85,B 0,C 180,E1 -12208.975,E2 -12208.975} C_VEL
LIN {X 0,Y 376.796,Z 725.073,A -85,B 0,C 180,E1 -12210.378,E2 -12210.378} C_VEL
LIN {X 0,Y 376.531,Z 730.393,A -85,B 0,C 180,E1 -12212.184,E2 -12212.184} C_VEL
LIN {X 0,Y 376.293,Z 733.804,A -85,B 0,C 180,E1 -12213.697,E2 -12213.697} C_VEL
LIN {X 0,Y 376.102,Z 736.949,A -85,B 0,C 180,E1 -12215.726,E2 -12215.726} C_VEL
LIN {X 0,Y 376.078,Z 738.095,A -85,B 0,C 180,E1 -12216.893,E2 -12216.893} C_VEL
LIN {X 0,Y 376.136,Z 738.696,A -85,B 0,C 180,E1 -12218.056,E2 -12218.056} C_VEL
LIN {X 0,Y 376.233,Z 738.857,A -85,B 0,C 180,E1 -12219.211,E2 -12219.211} C_VEL
LIN {X 0,Y 376.364,Z 738.519,A -85,B 0,C 180,E1 -12220.359,E2 -12220.359} C_VEL
LIN {X 0,Y 376.643,Z 737.093,A -85,B 0,C 180,E1 -12222.102,E2 -12222.102} C_VEL
LIN {X 0,Y 377.232,Z 733.621,A -85,B 0,C 180,E1 -12224.327,E2 -12224.327} C_VEL
LIN {X 0,Y 377.785,Z 729.654,A -85,B 0,C 180,E1 -12226.005,E2 -12226.005} C_VEL
LIN {X 0,Y 378.612,Z 723.441,A -85,B 0,C 180,E1 -12227.946,E2 -12227.946} C_VEL
LIN {X 0,Y 379.484,Z 716.525,A -85,B 0,C 180,E1 -12229.604,E2 -12229.604} C_VEL
LIN {X 0,Y 380.435,Z 707.881,A -85,B 0,C 180,E1 -12231.233,E2 -12231.233} C_VEL
LIN {X 0,Y 381.347,Z 698.944,A -85,B 0,C 180,E1 -12232.588,E2 -12232.588} C_VEL
LIN {X 0,Y 382.163,Z 689.193,A -85,B 0,C 180,E1 -12233.783,E2 -12233.783} C_VEL
LIN {X 0,Y 382.984,Z 678.101,A -85,B 0,C 180,E1 -12234.867,E2 -12234.867} C_VEL
LIN {X 0,Y 383.559,Z 667.921,A -85,B 0,C 180,E1 -12235.665,E2 -12235.665} C_VEL
LIN {X 0,Y 384.017,Z 655.996,A -85,B 0,C 180,E1 -12236.393,E2 -12236.393} C_VEL
LIN {X 0,Y 384.24,Z 643.201,A -85,B 0,C 180,E1 -12236.947,E2 -12236.947} C_VEL
LIN {X 0,Y 384.277,Z 625.036,A -85,B 0,C 180,E1 -12237.441,E2 -12237.441} C_VEL
LIN {X 0,Y 385.642,Z 574.672,A -85,B 0,C 180,E1 -12238.615,E2 -12238.615} C_VEL
LIN {X 0,Y 380.609,Z 562.906,A -85,B 0,C 180,E1 -12239.323,E2 -12239.323} C_VEL
LIN {X 0,Y 376.661,Z 554.682,A -85,B 0,C 180,E1 -12239.88,E2 -12239.88} C_VEL
LIN {X 0,Y 376.465,Z 553.594,A -85,B 0,C 180,E1 -12239.94,E2 -12239.94} C_VEL
LIN {X 0,Y 376.344,Z 553.608,A -85,B 0,C 180,E1 -12242.14,E2 -12242.14} C_VEL
LIN {X 0,Y 376.244,Z 553.621,A -85,B 0,C 180,E1 -12246.435,E2 -12246.435} C_VEL
LIN {X 0,Y 376.196,Z 553.625,A -85,B 0,C 180,E1 -12248.595,E2 -12248.595} C_VEL
LIN {X 0,Y 376.049,Z 553.642,A -85,B 0,C 180,E1 -12251.863,E2 -12251.863} C_VEL
LIN {X 0,Y 376.049,Z 553.637,A -85,B 0,C 180,E1 -12255.168,E2 -12255.168} C_VEL
LIN {X 0,Y 376.014,Z 553.648,A -85,B 0,C 180,E1 -12258.527,E2 -12258.527} C_VEL
LIN {X 0,Y 375.953,Z 553.654,A -85,B 0,C 180,E1 -12261.955,E2 -12261.955} C_VEL
LIN {X 0,Y 375.997,Z 553.648,A -85,B 0,C 180,E1 -12265.462,E2 -12265.462} C_VEL
LIN {X 0,Y 375.968,Z 553.653,A -85,B 0,C 180,E1 -12269.079,E2 -12269.079} C_VEL
LIN {X 0,Y 375.941,Z 553.658,A -85,B 0,C 180,E1 -12272.829,E2 -12272.829} C_VEL
LIN {X 0,Y 375.951,Z 553.654,A -85,B 0,C 180,E1 -12275.416,E2 -12275.416} C_VEL
LIN {X 0,Y 375.971,Z 553.65,A -85,B 0,C 180,E1 -12278.272,E2 -12278.272} C_VEL
LIN {X 0,Y 375.983,Z 553.653,A -85,B 0,C 180,E1 -12281.611,E2 -12281.611} C_VEL
LIN {X 0,Y 376.01,Z 553.647,A -85,B 0,C 180,E1 -12285.256,E2 -12285.256} C_VEL
LIN {X 0,Y 375.995,Z 553.649,A -85,B 0,C 180,E1 -12289.142,E2 -12289.142} C_VEL
LIN {X 0,Y 375.969,Z 553.654,A -85,B 0,C 180,E1 -12291.914,E2 -12291.914} C_VEL
LIN {X 0,Y 376,Z 553.815,A -85,B 0,C 180,E1 -12294.138,E2 -12294.138} C_VEL
LIN {X 0,Y 378.76,Z 563.862,A -85,B 0,C 180,E1 -12296.615,E2 -12296.615} C_VEL
LIN {X 0,Y 381.455,Z 575.42,A -85,B 0,C 180,E1 -12299.211,E2 -12299.211} C_VEL
LIN {X 0,Y 382.437,Z 580.383,A -85,B 0,C 180,E1 -12300.254,E2 -12300.254} C_VEL
LIN {X 0,Y 381.906,Z 586.668,A -85,B 0,C 180,E1 -12301.416,E2 -12301.416} C_VEL
LIN {X 0,Y 379.721,Z 608.152,A -85,B 0,C 180,E1 -12305.22,E2 -12305.22} C_VEL
LIN {X 0,Y 378.446,Z 623.307,A -85,B 0,C 180,E1 -12307.824,E2 -12307.824} C_VEL
LIN {X 0,Y 381.602,Z 645.98,A -85,B 0,C 180,E1 -12308.639,E2 -12308.639} C_VEL
LIN {X 0,Y 383.914,Z 673.693,A -85,B 0,C 180,E1 -12309.487,E2 -12309.487} C_VEL
LIN {X 0,Y 382.319,Z 736.974,A -85,B 0,C 180,E1 -12310.923,E2 -12310.923} C_VEL
LIN {X 0,Y 381.933,Z 746.025,A -85,B 0,C 180,E1 -12311.216,E2 -12311.216} C_VEL
LIN {X 0,Y 381.574,Z 759.98,A -85,B 0,C 180,E1 -12311.546,E2 -12311.546} C_VEL
LIN {X 0,Y 380.918,Z 773.023,A -85,B 0,C 180,E1 -12312.069,E2 -12312.069} C_VEL
LIN {X 0,Y 380.175,Z 785.423,A -85,B 0,C 180,E1 -12312.797,E2 -12312.797} C_VEL
LIN {X 0,Y 379.256,Z 797.324,A -85,B 0,C 180,E1 -12313.724,E2 -12313.724} C_VEL
LIN {X 0,Y 378.332,Z 807.911,A -85,B 0,C 180,E1 -12314.789,E2 -12314.789} C_VEL
LIN {X 0,Y 377.417,Z 817.563,A -85,B 0,C 180,E1 -12315.992,E2 -12315.992} C_VEL
LIN {X 0,Y 376.649,Z 826.354,A -85,B 0,C 180,E1 -12317.336,E2 -12317.336} C_VEL
LIN {X 0,Y 375.927,Z 833.59,A -85,B 0,C 180,E1 -12318.681,E2 -12318.681} C_VEL
LIN {X 0,Y 375.361,Z 840.682,A -85,B 0,C 180,E1 -12320.3,E2 -12320.3} C_VEL
LIN {X 0,Y 374.956,Z 846.315,A -85,B 0,C 180,E1 -12321.92,E2 -12321.92} C_VEL
LIN {X 0,Y 374.701,Z 851.253,A -85,B 0,C 180,E1 -12323.766,E2 -12323.766} C_VEL
LIN {X 0,Y 374.638,Z 854.954,A -85,B 0,C 180,E1 -12325.698,E2 -12325.698} C_VEL
LIN {X 0,Y 374.552,Z 856.382,A -85,B 0,C 180,E1 -12326.774,E2 -12326.774} C_VEL
LIN {X 0,Y 374.591,Z 857.391,A -85,B 0,C 180,E1 -12327.85,E2 -12327.85} C_VEL
LIN {X 0,Y 374.652,Z 858.008,A -85,B 0,C 180,E1 -12328.926,E2 -12328.926} C_VEL
LIN {X 0,Y 374.663,Z 858.227,A -85,B 0,C 180,E1 -12330.001,E2 -12330.001} C_VEL
LIN {X 0,Y 374.628,Z 858.003,A -85,B 0,C 180,E1 -12331.076,E2 -12331.076} C_VEL
LIN {X 0,Y 374.585,Z 857.383,A -85,B 0,C 180,E1 -12332.151,E2 -12332.151} C_VEL
LIN {X 0,Y 374.542,Z 856.37,A -85,B 0,C 180,E1 -12333.228,E2 -12333.228} C_VEL
LIN {X 0,Y 374.626,Z 854.937,A -85,B 0,C 180,E1 -12334.304,E2 -12334.304} C_VEL
LIN {X 0,Y 374.701,Z 851.234,A -85,B 0,C 180,E1 -12336.234,E2 -12336.234} C_VEL
LIN {X 0,Y 374.95,Z 846.286,A -85,B 0,C 180,E1 -12338.082,E2 -12338.082} C_VEL
LIN {X 0,Y 375.353,Z 840.64,A -85,B 0,C 180,E1 -12339.702,E2 -12339.702} C_VEL
LIN {X 0,Y 375.895,Z 833.532,A -85,B 0,C 180,E1 -12341.322,E2 -12341.322} C_VEL
LIN {X 0,Y 376.792,Z 824.672,A -85,B 0,C 180,E1 -12342.935,E2 -12342.935} C_VEL
LIN {X 0,Y 377.594,Z 815.687,A -85,B 0,C 180,E1 -12344.259,E2 -12344.259} C_VEL
LIN {X 0,Y 378.475,Z 805.376,A -85,B 0,C 180,E1 -12345.483,E2 -12345.483} C_VEL
LIN {X 0,Y 379.475,Z 794.077,A -85,B 0,C 180,E1 -12346.545,E2 -12346.545} C_VEL
LIN {X 0,Y 380.413,Z 782.304,A -85,B 0,C 180,E1 -12347.402,E2 -12347.402} C_VEL
LIN {X 0,Y 381.042,Z 770.739,A -85,B 0,C 180,E1 -12348.031,E2 -12348.031} C_VEL
LIN {X 0,Y 381.644,Z 757.411,A -85,B 0,C 180,E1 -12348.522,E2 -12348.522} C_VEL
LIN {X 0,Y 382.119,Z 734.653,A -85,B 0,C 180,E1 -12348.985,E2 -12348.985} C_VEL
LIN {X 0,Y 382.888,Z 674.627,A -85,B 0,C 180,E1 -12350.109,E2 -12350.109} C_VEL
LIN {X 0,Y 378.747,Z 638.938,A -85,B 0,C 180,E1 -12351.042,E2 -12351.042} C_VEL
LIN {X 0,Y 378.376,Z 635.863,A -85,B 0,C 180,E1 -12351.165,E2 -12351.165} C_VEL
LIN {X 0,Y 377.661,Z 627.089,A -85,B 0,C 180,E1 -12351.683,E2 -12351.683} C_VEL
LIN {X 0,Y 379.039,Z 607.958,A -85,B 0,C 180,E1 -12355.243,E2 -12355.243} C_VEL
LIN {X 0,Y 380.757,Z 588.106,A -85,B 0,C 180,E1 -12358.982,E2 -12358.982} C_VEL
LIN {X 0,Y 381.458,Z 578.865,A -85,B 0,C 180,E1 -12360.748,E2 -12360.748} C_VEL
LIN {X 0,Y 378.668,Z 565.605,A -85,B 0,C 180,E1 -12363.539,E2 -12363.539} C_VEL
LIN {X 0,Y 376.011,Z 553.648,A -85,B 0,C 180,E1 -12366.177,E2 -12366.177} C_VEL
LIN {X 0,Y 375.991,Z 553.649,A -85,B 0,C 180,E1 -12369.971,E2 -12369.971} C_VEL
LIN {X 0,Y 375.932,Z 553.647,A -85,B 0,C 180,E1 -12373.766,E2 -12373.766} C_VEL
LIN {X 0,Y 375.937,Z 553.658,A -85,B 0,C 180,E1 -12376.81,E2 -12376.81} C_VEL
LIN {X 0,Y 375.965,Z 553.651,A -85,B 0,C 180,E1 -12380.538,E2 -12380.538} C_VEL
LIN {X 0,Y 375.966,Z 553.643,A -85,B 0,C 180,E1 -12383.495,E2 -12383.495} C_VEL
LIN {X 0,Y 375.961,Z 553.652,A -85,B 0,C 180,E1 -12385.889,E2 -12385.889} C_VEL
LIN {X 0,Y 375.965,Z 553.643,A -85,B 0,C 180,E1 -12389.687,E2 -12389.687} C_VEL
LIN {X 0,Y 375.997,Z 553.647,A -85,B 0,C 180,E1 -12392.141,E2 -12392.141} C_VEL
LIN {X 0,Y 376.007,Z 553.637,A -85,B 0,C 180,E1 -12394.539,E2 -12394.539} C_VEL
LIN {X 0,Y 375.959,Z 553.652,A -85,B 0,C 180,E1 -12398.045,E2 -12398.045} C_VEL
LIN {X 0,Y 376.01,Z 553.631,A -85,B 0,C 180,E1 -12401.473,E2 -12401.473} C_VEL
LIN {X 0,Y 376.059,Z 553.637,A -85,B 0,C 180,E1 -12404.833,E2 -12404.833} C_VEL
LIN {X 0,Y 376.05,Z 553.63,A -85,B 0,C 180,E1 -12408.137,E2 -12408.137} C_VEL
LIN {X 0,Y 376.22,Z 553.619,A -85,B 0,C 180,E1 -12411.919,E2 -12411.919} C_VEL
LIN {X 0,Y 376.171,Z 553.623,A -85,B 0,C 180,E1 -12414.64,E2 -12414.64} C_VEL
LIN {X 0,Y 376.352,Z 553.587,A -85,B 0,C 180,E1 -12417.86,E2 -12417.86} C_VEL
LIN {X 0,Y 376.487,Z 553.589,A -85,B 0,C 180,E1 -12420,E2 -12420} C_VEL
LIN {X 0,Y 376.186,Z 553.621,A -85,B 0,C 180,E1 -12423.213,E2 -12423.213} C_VEL
LIN {X 0,Y 376.227,Z 553.612,A -85,B 0,C 180,E1 -12426.615,E2 -12426.615} C_VEL
LIN {X 0,Y 376.122,Z 553.634,A -85,B 0,C 180,E1 -12429.681,E2 -12429.681} C_VEL
LIN {X 0,Y 376.09,Z 553.624,A -85,B 0,C 180,E1 -12433.658,E2 -12433.658} C_VEL
LIN {X 0,Y 376.044,Z 553.639,A -85,B 0,C 180,E1 -12437.607,E2 -12437.607} C_VEL
LIN {X 0,Y 375.979,Z 553.645,A -85,B 0,C 180,E1 -12440.832,E2 -12440.832} C_VEL
LIN {X 0,Y 375.995,Z 553.639,A -85,B 0,C 180,E1 -12444.282,E2 -12444.282} C_VEL
LIN {X 0,Y 376.021,Z 553.643,A -85,B 0,C 180,E1 -12446.652,E2 -12446.652} C_VEL
LIN {X 0,Y 375.966,Z 553.643,A -85,B 0,C 180,E1 -12450.313,E2 -12450.313} C_VEL
LIN {X 0,Y 375.962,Z 553.654,A -85,B 0,C 180,E1 -12454.111,E2 -12454.111} C_VEL
LIN {X 0,Y 375.955,Z 553.656,A -85,B 0,C 180,E1 -12456.741,E2 -12456.741} C_VEL
LIN {X 0,Y 375.99,Z 553.646,A -85,B 0,C 180,E1 -12459.971,E2 -12459.971} C_VEL
LIN {X 0,Y 375.931,Z 553.652,A -85,B 0,C 180,E1 -12463.766,E2 -12463.766} C_VEL
LIN {X 0,Y 375.936,Z 553.639,A -85,B 0,C 180,E1 -12466.811,E2 -12466.811} C_VEL
LIN {X 0,Y 375.966,Z 553.651,A -85,B 0,C 180,E1 -12470.537,E2 -12470.537} C_VEL
LIN {X 0,Y 375.967,Z 553.653,A -85,B 0,C 180,E1 -12473.495,E2 -12473.495} C_VEL
LIN {X 0,Y 376.009,Z 553.786,A -85,B 0,C 180,E1 -12477.017,E2 -12477.017} C_VEL
LIN {X 0,Y 379.603,Z 567.61,A -85,B 0,C 180,E1 -12479.701,E2 -12479.701} C_VEL
LIN {X 0,Y 382.221,Z 579.626,A -85,B 0,C 180,E1 -12481.957,E2 -12481.957} C_VEL
LIN {X 0,Y 382.425,Z 583.602,A -85,B 0,C 180,E1 -12482.649,E2 -12482.649} C_VEL
LIN {X 0,Y 380.994,Z 604.719,A -85,B 0,C 180,E1 -12486.057,E2 -12486.057} C_VEL
LIN {X 0,Y 380.145,Z 623.308,A -85,B 0,C 180,E1 -12488.903,E2 -12488.903} C_VEL
LIN {X 0,Y 383.827,Z 646.877,A -85,B 0,C 180,E1 -12489.589,E2 -12489.589} C_VEL
LIN {X 0,Y 382.454,Z 735,A -85,B 0,C 180,E1 -12491.276,E2 -12491.276} C_VEL
LIN {X 0,Y 381.92,Z 748.166,A -85,B 0,C 180,E1 -12491.735,E2 -12491.735} C_VEL
LIN {X 0,Y 381.13,Z 761.165,A -85,B 0,C 180,E1 -12492.424,E2 -12492.424} C_VEL
LIN {X 0,Y 380.274,Z 773.872,A -85,B 0,C 180,E1 -12493.353,E2 -12493.353} C_VEL
LIN {X 0,Y 379.433,Z 784.105,A -85,B 0,C 180,E1 -12494.32,E2 -12494.32} C_VEL
LIN {X 0,Y 378.5,Z 795.085,A -85,B 0,C 180,E1 -12495.62,E2 -12495.62} C_VEL
LIN {X 0,Y 377.608,Z 803.353,A -85,B 0,C 180,E1 -12496.82,E2 -12496.82} C_VEL
LIN {X 0,Y 376.828,Z 810.977,A -85,B 0,C 180,E1 -12498.161,E2 -12498.161} C_VEL
LIN {X 0,Y 376.064,Z 818.416,A -85,B 0,C 180,E1 -12499.773,E2 -12499.773} C_VEL
LIN {X 0,Y 375.439,Z 824.391,A -85,B 0,C 180,E1 -12501.386,E2 -12501.386} C_VEL
LIN {X 0,Y 375.08,Z 829.765,A -85,B 0,C 180,E1 -12503.258,E2 -12503.258} C_VEL
LIN {X 0,Y 374.847,Z 832.723,A -85,B 0,C 180,E1 -12504.62,E2 -12504.62} C_VEL
LIN {X 0,Y 374.668,Z 834.585,A -85,B 0,C 180,E1 -12505.696,E2 -12505.696} C_VEL
LIN {X 0,Y 374.577,Z 836.006,A -85,B 0,C 180,E1 -12506.772,E2 -12506.772} C_VEL
LIN {X 0,Y 374.545,Z 837.616,A -85,B 0,C 180,E1 -12508.924,E2 -12508.924} C_VEL
LIN {X 0,Y 374.555,Z 837.85,A -85,B 0,C 180,E1 -12509.999,E2 -12509.999} C_VEL
LIN {X 0,Y 374.545,Z 837.659,A -85,B 0,C 180,E1 -12511.074,E2 -12511.074} C_VEL
LIN {X 0,Y 374.566,Z 836.11,A -85,B 0,C 180,E1 -12513.226,E2 -12513.226} C_VEL
LIN {X 0,Y 374.666,Z 834.745,A -85,B 0,C 180,E1 -12514.302,E2 -12514.302} C_VEL
LIN {X 0,Y 374.922,Z 831.873,A -85,B 0,C 180,E1 -12515.917,E2 -12515.917} C_VEL
LIN {X 0,Y 375.158,Z 827.972,A -85,B 0,C 180,E1 -12517.534,E2 -12517.534} C_VEL
LIN {X 0,Y 375.612,Z 822.92,A -85,B 0,C 180,E1 -12519.15,E2 -12519.15} C_VEL
LIN {X 0,Y 376.233,Z 816.403,A -85,B 0,C 180,E1 -12520.799,E2 -12520.799} C_VEL
LIN {X 0,Y 375.914,Z 813.086,A -85,B 0,C 180,E1 -12521.542,E2 -12521.542} C_VEL
LIN {X 0,Y 373.743,Z 807.405,A -85,B 0,C 180,E1 -12522.744,E2 -12522.744} C_VEL
LIN {X 0,Y 371.659,Z 801.172,A -85,B 0,C 180,E1 -12523.883,E2 -12523.883} C_VEL
LIN {X 0,Y 371.466,Z 796.953,A -85,B 0,C 180,E1 -12524.519,E2 -12524.519} C_VEL
LIN {X 0,Y 372.348,Z 787.558,A -85,B 0,C 180,E1 -12525.715,E2 -12525.715} C_VEL
LIN {X 0,Y 373.273,Z 776.67,A -85,B 0,C 180,E1 -12526.826,E2 -12526.826} C_VEL
LIN {X 0,Y 374.205,Z 764.828,A -85,B 0,C 180,E1 -12527.769,E2 -12527.769} C_VEL
LIN {X 0,Y 375.056,Z 752.482,A -85,B 0,C 180,E1 -12528.504,E2 -12528.504} C_VEL
LIN {X 0,Y 375.589,Z 740.486,A -85,B 0,C 180,E1 -12529.007,E2 -12529.007} C_VEL
LIN {X 0,Y 375.951,Z 725.882,A -85,B 0,C 180,E1 -12529.378,E2 -12529.378} C_VEL
LIN {X 0,Y 377.125,Z 649.231,A -85,B 0,C 180,E1 -12530.846,E2 -12530.846} C_VEL
LIN {X 0,Y 372.827,Z 624.275,A -85,B 0,C 180,E1 -12531.616,E2 -12531.616} C_VEL
LIN {X 0,Y 373.818,Z 604.727,A -85,B 0,C 180,E1 -12534.996,E2 -12534.996} C_VEL
LIN {X 0,Y 375.004,Z 587.01,A -85,B 0,C 180,E1 -12538.256,E2 -12538.256} C_VEL
LIN {X 0,Y 375.244,Z 582.33,A -85,B 0,C 180,E1 -12539.139,E2 -12539.139} C_VEL
LIN {X 0,Y 373.137,Z 571.437,A -85,B 0,C 180,E1 -12541.411,E2 -12541.411} C_VEL
LIN {X 0,Y 370.128,Z 559.135,A -85,B 0,C 180,E1 -12544.064,E2 -12544.064} C_VEL
LIN {X 0,Y 368.936,Z 554.532,A -85,B 0,C 180,E1 -12545.103,E2 -12545.103} C_VEL
LIN {X 0,Y 368.9,Z 554.527,A -85,B 0,C 180,E1 -12548.952,E2 -12548.952} C_VEL
LIN {X 0,Y 368.878,Z 554.534,A -85,B 0,C 180,E1 -12552.008,E2 -12552.008} C_VEL
LIN {X 0,Y 368.949,Z 554.522,A -85,B 0,C 180,E1 -12555.186,E2 -12555.186} C_VEL
LIN {X 0,Y 369.014,Z 554.52,A -85,B 0,C 180,E1 -12557.793,E2 -12557.793} C_VEL
LIN {X 0,Y 375.246,Z 572.47,A -85,B 0,C 180,E1 -12558.515,E2 -12558.515} C_VEL
LIN {X 0,Y 374.354,Z 634.036,A -85,B 0,C 180,E1 -12559.896,E2 -12559.896} C_VEL
LIN {X 0,Y 374.245,Z 647.583,A -85,B 0,C 180,E1 -12560.399,E2 -12560.399} C_VEL
LIN {X 0,Y 373.863,Z 661.248,A -85,B 0,C 180,E1 -12561.142,E2 -12561.142} C_VEL
LIN {X 0,Y 373.332,Z 673.378,A -85,B 0,C 180,E1 -12562.039,E2 -12562.039} C_VEL
LIN {X 0,Y 372.727,Z 685.829,A -85,B 0,C 180,E1 -12563.225,E2 -12563.225} C_VEL
LIN {X 0,Y 372.003,Z 696.748,A -85,B 0,C 180,E1 -12564.547,E2 -12564.547} C_VEL
LIN {X 0,Y 371.342,Z 706.374,A -85,B 0,C 180,E1 -12565.987,E2 -12565.987} C_VEL
LIN {X 0,Y 370.656,Z 715.126,A -85,B 0,C 180,E1 -12567.612,E2 -12567.612} C_VEL
LIN {X 0,Y 370.035,Z 723.046,A -85,B 0,C 180,E1 -12569.465,E2 -12569.465} C_VEL
LIN {X 0,Y 369.664,Z 728.195,A -85,B 0,C 180,E1 -12570.988,E2 -12570.988} C_VEL
LIN {X 0,Y 369.375,Z 733.034,A -85,B 0,C 180,E1 -12572.829,E2 -12572.829} C_VEL
LIN {X 0,Y 369.207,Z 735.449,A -85,B 0,C 180,E1 -12574.035,E2 -12574.035} C_VEL
LIN {X 0,Y 369.074,Z 738.343,A -85,B 0,C 180,E1 -12576.064,E2 -12576.064} C_VEL
LIN {X 0,Y 369.096,Z 739.546,A -85,B 0,C 180,E1 -12577.615,E2 -12577.615} C_VEL
LIN {X 0,Y 369.182,Z 739.899,A -85,B 0,C 180,E1 -12578.87,E2 -12578.87} C_VEL
LIN {X 0,Y 369.309,Z 739.77,A -85,B 0,C 180,E1 -12579.968,E2 -12579.968} C_VEL
LIN {X 0,Y 369.618,Z 738.525,A -85,B 0,C 180,E1 -12581.93,E2 -12581.93} C_VEL
LIN {X 0,Y 370.146,Z 735.627,A -85,B 0,C 180,E1 -12584.019,E2 -12584.019} C_VEL
LIN {X 0,Y 370.702,Z 732.016,A -85,B 0,C 180,E1 -12585.732,E2 -12585.732} C_VEL
LIN {X 0,Y 371.449,Z 727.178,A -85,B 0,C 180,E1 -12587.433,E2 -12587.433} C_VEL
LIN {X 0,Y 372.315,Z 720.992,A -85,B 0,C 180,E1 -12589.119,E2 -12589.119} C_VEL
LIN {X 0,Y 373.231,Z 713.173,A -85,B 0,C 180,E1 -12590.79,E2 -12590.79} C_VEL
LIN {X 0,Y 374.179,Z 705.123,A -85,B 0,C 180,E1 -12592.173,E2 -12592.173} C_VEL
LIN {X 0,Y 375.112,Z 695.38,A -85,B 0,C 180,E1 -12593.545,E2 -12593.545} C_VEL
LIN {X 0,Y 376.085,Z 684.314,A -85,B 0,C 180,E1 -12594.773,E2 -12594.773} C_VEL
LIN {X 0,Y 376.788,Z 673.635,A -85,B 0,C 180,E1 -12595.721,E2 -12595.721} C_VEL
LIN {X 0,Y 377.399,Z 661.89,A -85,B 0,C 180,E1 -12596.53,E2 -12596.53} C_VEL
LIN {X 0,Y 377.759,Z 648.544,A -85,B 0,C 180,E1 -12597.201,E2 -12597.201} C_VEL
LIN {X 0,Y 377.823,Z 635.559,A -85,B 0,C 180,E1 -12597.635,E2 -12597.635} C_VEL
LIN {X 0,Y 378.786,Z 591.9,A -85,B 0,C 180,E1 -12598.69,E2 -12598.69} C_VEL
LIN {X 0,Y 379.247,Z 576.547,A -85,B 0,C 180,E1 -12599.064,E2 -12599.064} C_VEL
LIN {X 0,Y 374.792,Z 566.163,A -85,B 0,C 180,E1 -12599.721,E2 -12599.721} C_VEL
LIN {X 0,Y 370.487,Z 557.5,A -85,B 0,C 180,E1 -12600.341,E2 -12600.341} C_VEL
LIN {X 0,Y 369.371,Z 554.722,A -85,B 0,C 180,E1 -12600.526,E2 -12600.526} C_VEL
LIN {X 0,Y 369.319,Z 554.485,A -85,B 0,C 180,E1 -12600.545,E2 -12600.545} C_VEL
LIN {X 0,Y 369.309,Z 554.485,A -85,B 0,C 180,E1 -12602.181,E2 -12602.181} C_VEL
LIN {X 0,Y 369.204,Z 554.497,A -85,B 0,C 180,E1 -12606.558,E2 -12606.558} C_VEL
LIN {X 0,Y 369.129,Z 554.508,A -85,B 0,C 180,E1 -12608.761,E2 -12608.761} C_VEL
LIN {X 0,Y 369.003,Z 554.52,A -85,B 0,C 180,E1 -12612.093,E2 -12612.093} C_VEL
LIN {X 0,Y 368.988,Z 554.515,A -85,B 0,C 180,E1 -12615.465,E2 -12615.465} C_VEL
LIN {X 0,Y 368.972,Z 554.526,A -85,B 0,C 180,E1 -12618.893,E2 -12618.893} C_VEL
LIN {X 0,Y 368.922,Z 554.532,A -85,B 0,C 180,E1 -12622.396,E2 -12622.396} C_VEL
LIN {X 0,Y 368.991,Z 554.52,A -85,B 0,C 180,E1 -12625.981,E2 -12625.981} C_VEL
LIN {X 0,Y 368.959,Z 554.527,A -85,B 0,C 180,E1 -12628.814,E2 -12628.814} C_VEL
LIN {X 0,Y 368.891,Z 554.535,A -85,B 0,C 180,E1 -12632.239,E2 -12632.239} C_VEL
LIN {X 0,Y 368.921,Z 554.526,A -85,B 0,C 180,E1 -12635.003,E2 -12635.003} C_VEL
LIN {X 0,Y 368.907,Z 554.533,A -85,B 0,C 180,E1 -12638.642,E2 -12638.642} C_VEL
LIN {X 0,Y 368.935,Z 554.531,A -85,B 0,C 180,E1 -12642.021,E2 -12642.021} C_VEL
LIN {X 0,Y 368.985,Z 554.522,A -85,B 0,C 180,E1 -12645.194,E2 -12645.194} C_VEL
LIN {X 0,Y 368.936,Z 554.531,A -85,B 0,C 180,E1 -12648.187,E2 -12648.187} C_VEL
LIN {X 0,Y 368.913,Z 554.535,A -85,B 0,C 180,E1 -12651.359,E2 -12651.359} C_VEL
LIN {X 0,Y 368.957,Z 554.7,A -85,B 0,C 180,E1 -12653.489,E2 -12653.489} C_VEL
LIN {X 0,Y 371.931,Z 565.368,A -85,B 0,C 180,E1 -12656.245,E2 -12656.245} C_VEL
LIN {X 0,Y 374.636,Z 577.002,A -85,B 0,C 180,E1 -12658.945,E2 -12658.945} C_VEL
LIN {X 0,Y 375.619,Z 581.725,A -85,B 0,C 180,E1 -12659.968,E2 -12659.968} C_VEL
LIN {X 0,Y 375.372,Z 586.443,A -85,B 0,C 180,E1 -12660.872,E2 -12660.872} C_VEL
LIN {X 0,Y 372.993,Z 607.752,A -85,B 0,C 180,E1 -12664.746,E2 -12664.746} C_VEL
LIN {X 0,Y 371.687,Z 621.75,A -85,B 0,C 180,E1 -12667.231,E2 -12667.231} C_VEL
LIN {X 0,Y 374.545,Z 641.642,A -85,B 0,C 180,E1 -12668.011,E2 -12668.011} C_VEL
LIN {X 0,Y 376.739,Z 664.112,A -85,B 0,C 180,E1 -12668.75,E2 -12668.75} C_VEL
LIN {X 0,Y 377.406,Z 676.728,A -85,B 0,C 180,E1 -12669.118,E2 -12669.118} C_VEL
LIN {X 0,Y 375.762,Z 735.91,A -85,B 0,C 180,E1 -12670.506,E2 -12670.506} C_VEL
LIN {X 0,Y 375.227,Z 747.765,A -85,B 0,C 180,E1 -12670.903,E2 -12670.903} C_VEL
LIN {X 0,Y 374.81,Z 760.941,A -85,B 0,C 180,E1 -12671.236,E2 -12671.236} C_VEL
LIN {X 0,Y 374.078,Z 774.154,A -85,B 0,C 180,E1 -12671.801,E2 -12671.801} C_VEL
LIN {X 0,Y 373.227,Z 787.212,A -85,B 0,C 180,E1 -12672.608,E2 -12672.608} C_VEL
LIN {X 0,Y 372.31,Z 798.576,A -85,B 0,C 180,E1 -12673.553,E2 -12673.553} C_VEL
LIN {X 0,Y 371.338,Z 808.898,A -85,B 0,C 180,E1 -12674.636,E2 -12674.636} C_VEL
LIN {X 0,Y 370.319,Z 819.315,A -85,B 0,C 180,E1 -12675.998,E2 -12675.998} C_VEL
LIN {X 0,Y 369.566,Z 827.732,A -85,B 0,C 180,E1 -12677.369,E2 -12677.369} C_VEL
LIN {X 0,Y 368.704,Z 835.925,A -85,B 0,C 180,E1 -12679.013,E2 -12679.013} C_VEL
LIN {X 0,Y 368.182,Z 842.51,A -85,B 0,C 180,E1 -12680.663,E2 -12680.663} C_VEL
LIN {X 0,Y 367.796,Z 847.739,A -85,B 0,C 180,E1 -12682.314,E2 -12682.314} C_VEL
LIN {X 0,Y 367.604,Z 851.423,A -85,B 0,C 180,E1 -12683.805,E2 -12683.805} C_VEL
LIN {X 0,Y 367.563,Z 854.762,A -85,B 0,C 180,E1 -12685.615,E2 -12685.615} C_VEL
LIN {X 0,Y 367.467,Z 856.189,A -85,B 0,C 180,E1 -12686.712,E2 -12686.712} C_VEL
LIN {X 0,Y 367.55,Z 857.815,A -85,B 0,C 180,E1 -12688.905,E2 -12688.905} C_VEL
LIN {X 0,Y 367.594,Z 858.035,A -85,B 0,C 180,E1 -12690.001,E2 -12690.001} C_VEL
LIN {X 0,Y 367.528,Z 857.81,A -85,B 0,C 180,E1 -12691.097,E2 -12691.097} C_VEL
LIN {X 0,Y 367.482,Z 857.189,A -85,B 0,C 180,E1 -12692.193,E2 -12692.193} C_VEL
LIN {X 0,Y 367.456,Z 856.177,A -85,B 0,C 180,E1 -12693.29,E2 -12693.29} C_VEL
LIN {X 0,Y 367.551,Z 854.744,A -85,B 0,C 180,E1 -12694.387,E2 -12694.387} C_VEL
LIN {X 0,Y 367.596,Z 851.429,A -85,B 0,C 180,E1 -12696.183,E2 -12696.183} C_VEL
LIN {X 0,Y 367.801,Z 847.709,A -85,B 0,C 180,E1 -12697.688,E2 -12697.688} C_VEL
LIN {X 0,Y 368.219,Z 841.457,A -85,B 0,C 180,E1 -12699.615,E2 -12699.615} C_VEL
LIN {X 0,Y 368.773,Z 834.637,A -85,B 0,C 180,E1 -12701.265,E2 -12701.265} C_VEL
LIN {X 0,Y 369.667,Z 826.103,A -85,B 0,C 180,E1 -12702.909,E2 -12702.909} C_VEL
LIN {X 0,Y 370.5,Z 817.311,A -85,B 0,C 180,E1 -12704.277,E2 -12704.277} C_VEL
LIN {X 0,Y 371.489,Z 806.462,A -85,B 0,C 180,E1 -12705.64,E2 -12705.64} C_VEL
LIN {X 0,Y 372.531,Z 795.466,A -85,B 0,C 180,E1 -12706.721,E2 -12706.721} C_VEL
LIN {X 0,Y 373.555,Z 783.13,A -85,B 0,C 180,E1 -12707.661,E2 -12707.661} C_VEL
LIN {X 0,Y 374.253,Z 771.325,A -85,B 0,C 180,E1 -12708.334,E2 -12708.334} C_VEL
LIN {X 0,Y 374.895,Z 758.383,A -85,B 0,C 180,E1 -12708.833,E2 -12708.833} C_VEL
LIN {X 0,Y 375.351,Z 741.761,A -85,B 0,C 180,E1 -12709.199,E2 -12709.199} C_VEL
LIN {X 0,Y 376.155,Z 674.711,A -85,B 0,C 180,E1 -12710.481,E2 -12710.481} C_VEL
LIN {X 0,Y 372.112,Z 639.848,A -85,B 0,C 180,E1 -12711.415,E2 -12711.415} C_VEL
LIN {X 0,Y 371.623,Z 635.707,A -85,B 0,C 180,E1 -12711.569,E2 -12711.569} C_VEL
LIN {X 0,Y 370.768,Z 625.402,A -85,B 0,C 180,E1 -12712.189,E2 -12712.189} C_VEL
LIN {X 0,Y 372.213,Z 606.727,A -85,B 0,C 180,E1 -12715.74,E2 -12715.74} C_VEL
LIN {X 0,Y 374.001,Z 586.881,A -85,B 0,C 180,E1 -12719.549,E2 -12719.549} C_VEL
LIN {X 0,Y 374.517,Z 580.68,A -85,B 0,C 180,E1 -12720.755,E2 -12720.755} C_VEL
LIN {X 0,Y 372.26,Z 569.239,A -85,B 0,C 180,E1 -12723.196,E2 -12723.196} C_VEL
LIN {X 0,Y 368.943,Z 554.529,A -85,B 0,C 180,E1 -12726.522,E2 -12726.522} C_VEL
LIN {X 0,Y 368.913,Z 554.531,A -85,B 0,C 180,E1 -12730.37,E2 -12730.37} C_VEL
LIN {X 0,Y 368.884,Z 554.525,A -85,B 0,C 180,E1 -12733.616,E2 -12733.616} C_VEL
LIN {X 0,Y 368.889,Z 554.535,A -85,B 0,C 180,E1 -12736.696,E2 -12736.696} C_VEL
LIN {X 0,Y 368.914,Z 554.531,A -85,B 0,C 180,E1 -12739.643,E2 -12739.643} C_VEL
LIN {X 0,Y 368.904,Z 554.522,A -85,B 0,C 180,E1 -12743.144,E2 -12743.144} C_VEL
LIN {X 0,Y 368.898,Z 554.531,A -85,B 0,C 180,E1 -12746.462,E2 -12746.462} C_VEL
LIN {X 0,Y 368.93,Z 554.516,A -85,B 0,C 180,E1 -12749.047,E2 -12749.047} C_VEL
LIN {X 0,Y 368.981,Z 554.525,A -85,B 0,C 180,E1 -12751.564,E2 -12751.564} C_VEL
LIN {X 0,Y 369.001,Z 554.51,A -85,B 0,C 180,E1 -12754.02,E2 -12754.02} C_VEL
LIN {X 0,Y 368.926,Z 554.529,A -85,B 0,C 180,E1 -12757.604,E2 -12757.604} C_VEL
LIN {X 0,Y 368.959,Z 554.514,A -85,B 0,C 180,E1 -12761.106,E2 -12761.106} C_VEL
LIN {X 0,Y 368.999,Z 554.515,A -85,B 0,C 180,E1 -12764.535,E2 -12764.535} C_VEL
LIN {X 0,Y 369.005,Z 554.509,A -85,B 0,C 180,E1 -12767.907,E2 -12767.907} C_VEL
LIN {X 0,Y 369.167,Z 554.497,A -85,B 0,C 180,E1 -12771.869,E2 -12771.869} C_VEL
LIN {X 0,Y 369.144,Z 554.498,A -85,B 0,C 180,E1 -12774.538,E2 -12774.538} C_VEL
LIN {X 0,Y 369.317,Z 554.462,A -85,B 0,C 180,E1 -12777.819,E2 -12777.819} C_VEL
LIN {X 0,Y 369.457,Z 554.464,A -85,B 0,C 180,E1 -12780,E2 -12780} C_VEL
LIN {X 0,Y 369.317,Z 554.477,A -85,B 0,C 180,E1 -12782.181,E2 -12782.181} C_VEL
LIN {X 0,Y 369.198,Z 554.487,A -85,B 0,C 180,E1 -12786.599,E2 -12786.599} C_VEL
LIN {X 0,Y 369.123,Z 554.503,A -85,B 0,C 180,E1 -12788.761,E2 -12788.761} C_VEL
LIN {X 0,Y 369.005,Z 554.501,A -85,B 0,C 180,E1 -12792.093,E2 -12792.093} C_VEL
LIN {X 0,Y 368.999,Z 554.519,A -85,B 0,C 180,E1 -12795.465,E2 -12795.465} C_VEL
LIN {X 0,Y 368.959,Z 554.509,A -85,B 0,C 180,E1 -12798.894,E2 -12798.894} C_VEL
LIN {X 0,Y 368.933,Z 554.529,A -85,B 0,C 180,E1 -12802.395,E2 -12802.395} C_VEL
LIN {X 0,Y 369.001,Z 554.509,A -85,B 0,C 180,E1 -12805.98,E2 -12805.98} C_VEL
LIN {X 0,Y 368.916,Z 554.528,A -85,B 0,C 180,E1 -12809.69,E2 -12809.69} C_VEL
LIN {X 0,Y 368.902,Z 554.533,A -85,B 0,C 180,E1 -12813.044,E2 -12813.044} C_VEL
LIN {X 0,Y 368.919,Z 554.527,A -85,B 0,C 180,E1 -12816.197,E2 -12816.197} C_VEL
LIN {X 0,Y 368.904,Z 554.529,A -85,B 0,C 180,E1 -12818.953,E2 -12818.953} C_VEL
LIN {X 0,Y 368.884,Z 554.538,A -85,B 0,C 180,E1 -12822.009,E2 -12822.009} C_VEL
LIN {X 0,Y 368.882,Z 554.534,A -85,B 0,C 180,E1 -12825.176,E2 -12825.176} C_VEL
LIN {X 0,Y 368.883,Z 554.518,A -85,B 0,C 180,E1 -12828.177,E2 -12828.177} C_VEL
LIN {X 0,Y 368.912,Z 554.523,A -85,B 0,C 180,E1 -12831.36,E2 -12831.36} C_VEL
LIN {X 0,Y 368.94,Z 554.53,A -85,B 0,C 180,E1 -12835.146,E2 -12835.146} C_VEL
LIN {X 0,Y 368.963,Z 554.71,A -85,B 0,C 180,E1 -12836.577,E2 -12836.577} C_VEL
LIN {X 0,Y 373.007,Z 570.149,A -85,B 0,C 180,E1 -12839.613,E2 -12839.613} C_VEL
LIN {X 0,Y 375.621,Z 582.254,A -85,B 0,C 180,E1 -12841.915,E2 -12841.915} C_VEL
LIN {X 0,Y 375.557,Z 586.943,A -85,B 0,C 180,E1 -12842.71,E2 -12842.71} C_VEL
LIN {X 0,Y 374.052,Z 608.255,A -85,B 0,C 180,E1 -12846.173,E2 -12846.173} C_VEL
LIN {X 0,Y 373.389,Z 623.459,A -85,B 0,C 180,E1 -12848.507,E2 -12848.507} C_VEL
LIN {X 0,Y 377.168,Z 647.21,A -85,B 0,C 180,E1 -12849.217,E2 -12849.217} C_VEL
LIN {X 0,Y 375.759,Z 735.128,A -85,B 0,C 180,E1 -12850.929,E2 -12850.929} C_VEL
LIN {X 0,Y 375.193,Z 748.328,A -85,B 0,C 180,E1 -12851.395,E2 -12851.395} C_VEL
LIN {X 0,Y 374.385,Z 761.338,A -85,B 0,C 180,E1 -12852.097,E2 -12852.097} C_VEL
LIN {X 0,Y 373.636,Z 772.439,A -85,B 0,C 180,E1 -12852.908,E2 -12852.908} C_VEL
LIN {X 0,Y 372.767,Z 782.342,A -85,B 0,C 180,E1 -12853.818,E2 -12853.818} C_VEL
LIN {X 0,Y 371.845,Z 793.201,A -85,B 0,C 180,E1 -12855.077,E2 -12855.077} C_VEL
LIN {X 0,Y 370.696,Z 803.543,A -85,B 0,C 180,E1 -12856.57,E2 -12856.57} C_VEL
LIN {X 0,Y 369.865,Z 811.168,A -85,B 0,C 180,E1 -12857.935,E2 -12857.935} C_VEL
LIN {X 0,Y 369.056,Z 818.608,A -85,B 0,C 180,E1 -12859.576,E2 -12859.576} C_VEL
LIN {X 0,Y 368.406,Z 824.584,A -85,B 0,C 180,E1 -12861.221,E2 -12861.221} C_VEL
LIN {X 0,Y 368.05,Z 829.307,A -85,B 0,C 180,E1 -12862.87,E2 -12862.87} C_VEL
LIN {X 0,Y 367.781,Z 832.917,A -85,B 0,C 180,E1 -12864.516,E2 -12864.516} C_VEL
LIN {X 0,Y 367.604,Z 834.778,A -85,B 0,C 180,E1 -12865.613,E2 -12865.613} C_VEL
LIN {X 0,Y 367.49,Z 836.2,A -85,B 0,C 180,E1 -12866.71,E2 -12866.71} C_VEL
LIN {X 0,Y 367.448,Z 837.809,A -85,B 0,C 180,E1 -12868.903,E2 -12868.903} C_VEL
LIN {X 0,Y 367.458,Z 838.043,A -85,B 0,C 180,E1 -12869.999,E2 -12869.999} C_VEL
LIN {X 0,Y 367.447,Z 837.852,A -85,B 0,C 180,E1 -12871.095,E2 -12871.095} C_VEL
LIN {X 0,Y 367.48,Z 836.302,A -85,B 0,C 180,E1 -12873.288,E2 -12873.288} C_VEL
LIN {X 0,Y 367.601,Z 834.936,A -85,B 0,C 180,E1 -12874.385,E2 -12874.385} C_VEL
LIN {X 0,Y 367.869,Z 831.629,A -85,B 0,C 180,E1 -12876.232,E2 -12876.232} C_VEL
LIN {X 0,Y 368.266,Z 826.593,A -85,B 0,C 180,E1 -12878.228,E2 -12878.228} C_VEL
LIN {X 0,Y 368.809,Z 821.143,A -85,B 0,C 180,E1 -12879.874,E2 -12879.874} C_VEL
LIN {X 0,Y 369.536,Z 814.308,A -85,B 0,C 180,E1 -12881.518,E2 -12881.518} C_VEL
LIN {X 0,Y 370.445,Z 805.741,A -85,B 0,C 180,E1 -12883.158,E2 -12883.158} C_VEL
LIN {X 0,Y 371.466,Z 796.953,A -85,B 0,C 180,E1 -12884.519,E2 -12884.519} C_VEL
LIN {X 0,Y 371.271,Z 792.599,A -85,B 0,C 180,E1 -12885.13,E2 -12885.13} C_VEL
LIN {X 0,Y 369.198,Z 785.307,A -85,B 0,C 180,E1 -12886.126,E2 -12886.126} C_VEL
LIN {X 0,Y 367.114,Z 777.636,A -85,B 0,C 180,E1 -12887.043,E2 -12887.043} C_VEL
LIN {X 0,Y 366.881,Z 772.598,A -85,B 0,C 180,E1 -12887.519,E2 -12887.519} C_VEL
LIN {X 0,Y 367.784,Z 760.898,A -85,B 0,C 180,E1 -12888.378,E2 -12888.378} C_VEL
LIN {X 0,Y 368.524,Z 748.387,A -85,B 0,C 180,E1 -12889.06,E2 -12889.06} C_VEL
LIN {X 0,Y 369.038,Z 736.37,A -85,B 0,C 180,E1 -12889.502,E2 -12889.502} C_VEL
LIN {X 0,Y 369.771,Z 698.046,A -85,B 0,C 180,E1 -12890.283,E2 -12890.283} C_VEL
LIN {X 0,Y 370.475,Z 649.822,A -85,B 0,C 180,E1 -12891.227,E2 -12891.227} C_VEL
LIN {X 0,Y 366.043,Z 624.433,A -85,B 0,C 180,E1 -12892.037,E2 -12892.037} C_VEL
LIN {X 0,Y 367.089,Z 605.132,A -85,B 0,C 180,E1 -12895.401,E2 -12895.401} C_VEL
LIN {X 0,Y 368.359,Z 587.054,A -85,B 0,C 180,E1 -12898.767,E2 -12898.767} C_VEL
LIN {X 0,Y 368.191,Z 582.024,A -85,B 0,C 180,E1 -12899.753,E2 -12899.753} C_VEL
LIN {X 0,Y 365.334,Z 568.835,A -85,B 0,C 180,E1 -12902.59,E2 -12902.59} C_VEL
LIN {X 0,Y 362.512,Z 557.919,A -85,B 0,C 180,E1 -12905.005,E2 -12905.005} C_VEL
LIN {X 0,Y 361.9,Z 555.403,A -85,B 0,C 180,E1 -12905.584,E2 -12905.584} C_VEL
LIN {X 0,Y 361.867,Z 555.402,A -85,B 0,C 180,E1 -12909.026,E2 -12909.026} C_VEL
LIN {X 0,Y 361.833,Z 555.4,A -85,B 0,C 180,E1 -12912.827,E2 -12912.827} C_VEL
LIN {X 0,Y 361.906,Z 555.405,A -85,B 0,C 180,E1 -12915.93,E2 -12915.93} C_VEL
LIN {X 0,Y 361.978,Z 555.545,A -85,B 0,C 180,E1 -12917.484,E2 -12917.484} C_VEL
LIN {X 0,Y 368.468,Z 574.052,A -85,B 0,C 180,E1 -12918.244,E2 -12918.244} C_VEL
LIN {X 0,Y 367.493,Z 635.506,A -85,B 0,C 180,E1 -12919.656,E2 -12919.656} C_VEL
LIN {X 0,Y 367.384,Z 649.072,A -85,B 0,C 180,E1 -12920.181,E2 -12920.181} C_VEL
LIN {X 0,Y 366.993,Z 661.74,A -85,B 0,C 180,E1 -12920.883,E2 -12920.883} C_VEL
LIN {X 0,Y 366.426,Z 674.559,A -85,B 0,C 180,E1 -12921.845,E2 -12921.845} C_VEL
LIN {X 0,Y 365.851,Z 685.863,A -85,B 0,C 180,E1 -12922.935,E2 -12922.935} C_VEL
LIN {X 0,Y 365.173,Z 696.296,A -85,B 0,C 180,E1 -12924.182,E2 -12924.182} C_VEL
LIN {X 0,Y 364.431,Z 706.244,A -85,B 0,C 180,E1 -12925.661,E2 -12925.661} C_VEL
LIN {X 0,Y 363.758,Z 714.932,A -85,B 0,C 180,E1 -12927.25,E2 -12927.25} C_VEL
LIN {X 0,Y 363.221,Z 721.913,A -85,B 0,C 180,E1 -12928.829,E2 -12928.829} C_VEL
LIN {X 0,Y 362.691,Z 728.426,A -85,B 0,C 180,E1 -12930.686,E2 -12930.686} C_VEL
LIN {X 0,Y 362.469,Z 732.76,A -85,B 0,C 180,E1 -12932.267,E2 -12932.267} C_VEL
LIN {X 0,Y 362.17,Z 736.595,A -85,B 0,C 180,E1 -12934.111,E2 -12934.111} C_VEL
LIN {X 0,Y 362.057,Z 739.192,A -85,B 0,C 180,E1 -12935.943,E2 -12935.943} C_VEL
LIN {X 0,Y 362.045,Z 740.266,A -85,B 0,C 180,E1 -12937.155,E2 -12937.155} C_VEL
LIN {X 0,Y 362.142,Z 740.943,A -85,B 0,C 180,E1 -12938.669,E2 -12938.669} C_VEL
LIN {X 0,Y 362.409,Z 740.57,A -85,B 0,C 180,E1 -12940.751,E2 -12940.751} C_VEL
LIN {X 0,Y 362.617,Z 739.733,A -85,B 0,C 180,E1 -12941.935,E2 -12941.935} C_VEL
LIN {X 0,Y 362.898,Z 738.42,A -85,B 0,C 180,E1 -12943.112,E2 -12943.112} C_VEL
LIN {X 0,Y 363.537,Z 734.931,A -85,B 0,C 180,E1 -12945.146,E2 -12945.146} C_VEL
LIN {X 0,Y 364.391,Z 729.826,A -85,B 0,C 180,E1 -12947.185,E2 -12947.185} C_VEL
LIN {X 0,Y 365.38,Z 723.083,A -85,B 0,C 180,E1 -12949.155,E2 -12949.155} C_VEL
LIN {X 0,Y 366.232,Z 716.766,A -85,B 0,C 180,E1 -12950.612,E2 -12950.612} C_VEL
LIN {X 0,Y 367.171,Z 709.298,A -85,B 0,C 180,E1 -12952.023,E2 -12952.023} C_VEL
LIN {X 0,Y 368.17,Z 700.19,A -85,B 0,C 180,E1 -12953.423,E2 -12953.423} C_VEL
LIN {X 0,Y 369.174,Z 690.047,A -85,B 0,C 180,E1 -12954.675,E2 -12954.675} C_VEL
LIN {X 0,Y 370.06,Z 678.898,A -85,B 0,C 180,E1 -12955.78,E2 -12955.78} C_VEL
LIN {X 0,Y 370.741,Z 667.292,A -85,B 0,C 180,E1 -12956.672,E2 -12956.672} C_VEL
LIN {X 0,Y 371.257,Z 653.668,A -85,B 0,C 180,E1 -12957.457,E2 -12957.457} C_VEL
LIN {X 0,Y 371.397,Z 640.668,A -85,B 0,C 180,E1 -12957.967,E2 -12957.967} C_VEL
LIN {X 0,Y 371.9,Z 611.451,A -85,B 0,C 180,E1 -12958.714,E2 -12958.714} C_VEL
LIN {X 0,Y 372.96,Z 578.426,A -85,B 0,C 180,E1 -12959.533,E2 -12959.533} C_VEL
LIN {X 0,Y 367.881,Z 567.031,A -85,B 0,C 180,E1 -12960.302,E2 -12960.302} C_VEL
LIN {X 0,Y 363.82,Z 559.015,A -85,B 0,C 180,E1 -12960.925,E2 -12960.925} C_VEL
LIN {X 0,Y 362.482,Z 556.568,A -85,B 0,C 180,E1 -12961.128,E2 -12961.128} C_VEL
LIN {X 0,Y 362.219,Z 555.368,A -85,B 0,C 180,E1 -12961.216,E2 -12961.216} C_VEL
LIN {X 0,Y 362.064,Z 555.384,A -85,B 0,C 180,E1 -12963.338,E2 -12963.338} C_VEL
LIN {X 0,Y 362.167,Z 555.372,A -85,B 0,C 180,E1 -12966.686,E2 -12966.686} C_VEL
LIN {X 0,Y 362.065,Z 555.386,A -85,B 0,C 180,E1 -12968.933,E2 -12968.933} C_VEL
LIN {X 0,Y 361.956,Z 555.395,A -85,B 0,C 180,E1 -12972.332,E2 -12972.332} C_VEL
LIN {X 0,Y 361.952,Z 555.399,A -85,B 0,C 180,E1 -12974.621,E2 -12974.621} C_VEL
LIN {X 0,Y 361.95,Z 555.398,A -85,B 0,C 180,E1 -12978.1,E2 -12978.1} C_VEL
LIN {X 0,Y 361.882,Z 555.406,A -85,B 0,C 180,E1 -12981.654,E2 -12981.654} C_VEL
LIN {X 0,Y 361.919,Z 555.402,A -85,B 0,C 180,E1 -12985.291,E2 -12985.291} C_VEL
LIN {X 0,Y 361.914,Z 555.4,A -85,B 0,C 180,E1 -12987.779,E2 -12987.779} C_VEL
LIN {X 0,Y 361.838,Z 555.414,A -85,B 0,C 180,E1 -12991.286,E2 -12991.286} C_VEL
LIN {X 0,Y 361.846,Z 555.408,A -85,B 0,C 180,E1 -12994.281,E2 -12994.281} C_VEL
LIN {X 0,Y 361.858,Z 555.406,A -85,B 0,C 180,E1 -12997.224,E2 -12997.224} C_VEL
LIN {X 0,Y 361.898,Z 555.404,A -85,B 0,C 180,E1 -13000.769,E2 -13000.769} C_VEL
LIN {X 0,Y 361.927,Z 555.405,A -85,B 0,C 180,E1 -13004.352,E2 -13004.352} C_VEL
LIN {X 0,Y 361.881,Z 555.408,A -85,B 0,C 180,E1 -13007.56,E2 -13007.56} C_VEL
LIN {X 0,Y 361.873,Z 555.409,A -85,B 0,C 180,E1 -13010.973,E2 -13010.973} C_VEL
LIN {X 0,Y 361.872,Z 555.474,A -85,B 0,C 180,E1 -13012.776,E2 -13012.776} C_VEL
LIN {X 0,Y 364.584,Z 564.903,A -85,B 0,C 180,E1 -13015.345,E2 -13015.345} C_VEL
LIN {X 0,Y 367.48,Z 576.896,A -85,B 0,C 180,E1 -13018.271,E2 -13018.271} C_VEL
LIN {X 0,Y 368.935,Z 584.776,A -85,B 0,C 180,E1 -13020.03,E2 -13020.03} C_VEL
LIN {X 0,Y 367.237,Z 598.744,A -85,B 0,C 180,E1 -13022.66,E2 -13022.66} C_VEL
LIN {X 0,Y 365.074,Z 619.313,A -85,B 0,C 180,E1 -13026.427,E2 -13026.427} C_VEL
LIN {X 0,Y 364.994,Z 620.8,A -85,B 0,C 180,E1 -13026.658,E2 -13026.658} C_VEL
LIN {X 0,Y 368.222,Z 642.573,A -85,B 0,C 180,E1 -13027.537,E2 -13027.537} C_VEL
LIN {X 0,Y 370.322,Z 664.779,A -85,B 0,C 180,E1 -13028.299,E2 -13028.299} C_VEL
LIN {X 0,Y 370.957,Z 677.75,A -85,B 0,C 180,E1 -13028.686,E2 -13028.686} C_VEL
LIN {X 0,Y 369.228,Z 735.375,A -85,B 0,C 180,E1 -13030.074,E2 -13030.074} C_VEL
LIN {X 0,Y 368.485,Z 749.451,A -85,B 0,C 180,E1 -13030.576,E2 -13030.576} C_VEL
LIN {X 0,Y 368.014,Z 762.627,A -85,B 0,C 180,E1 -13030.948,E2 -13030.948} C_VEL
LIN {X 0,Y 367.263,Z 775.283,A -85,B 0,C 180,E1 -13031.523,E2 -13031.523} C_VEL
LIN {X 0,Y 366.45,Z 787.046,A -85,B 0,C 180,E1 -13032.276,E2 -13032.276} C_VEL
LIN {X 0,Y 365.471,Z 798.401,A -85,B 0,C 180,E1 -13033.236,E2 -13033.236} C_VEL
LIN {X 0,Y 364.471,Z 808.718,A -85,B 0,C 180,E1 -13034.339,E2 -13034.339} C_VEL
LIN {X 0,Y 363.41,Z 819.131,A -85,B 0,C 180,E1 -13035.726,E2 -13035.726} C_VEL
LIN {X 0,Y 362.589,Z 827.544,A -85,B 0,C 180,E1 -13037.122,E2 -13037.122} C_VEL
LIN {X 0,Y 361.689,Z 835.736,A -85,B 0,C 180,E1 -13038.797,E2 -13038.797} C_VEL
LIN {X 0,Y 361.122,Z 842.319,A -85,B 0,C 180,E1 -13040.479,E2 -13040.479} C_VEL
LIN {X 0,Y 360.729,Z 847.548,A -85,B 0,C 180,E1 -13042.163,E2 -13042.163} C_VEL
LIN {X 0,Y 360.522,Z 851.542,A -85,B 0,C 180,E1 -13043.823,E2 -13043.823} C_VEL
LIN {X 0,Y 360.468,Z 854.57,A -85,B 0,C 180,E1 -13045.528,E2 -13045.528} C_VEL
LIN {X 0,Y 360.384,Z 855.997,A -85,B 0,C 180,E1 -13046.647,E2 -13046.647} C_VEL
LIN {X 0,Y 360.449,Z 857.622,A -85,B 0,C 180,E1 -13048.884,E2 -13048.884} C_VEL
LIN {X 0,Y 360.508,Z 857.842,A -85,B 0,C 180,E1 -13050.001,E2 -13050.001} C_VEL
LIN {X 0,Y 360.428,Z 857.616,A -85,B 0,C 180,E1 -13051.118,E2 -13051.118} C_VEL
LIN {X 0,Y 360.374,Z 855.984,A -85,B 0,C 180,E1 -13053.355,E2 -13053.355} C_VEL
LIN {X 0,Y 360.457,Z 854.55,A -85,B 0,C 180,E1 -13054.474,E2 -13054.474} C_VEL
LIN {X 0,Y 360.493,Z 851.613,A -85,B 0,C 180,E1 -13056.133,E2 -13056.133} C_VEL
LIN {X 0,Y 360.731,Z 847.516,A -85,B 0,C 180,E1 -13057.839,E2 -13057.839} C_VEL
LIN {X 0,Y 361.19,Z 841.264,A -85,B 0,C 180,E1 -13059.804,E2 -13059.804} C_VEL
LIN {X 0,Y 361.789,Z 834.446,A -85,B 0,C 180,E1 -13061.486,E2 -13061.486} C_VEL
LIN {X 0,Y 362.73,Z 825.913,A -85,B 0,C 180,E1 -13063.16,E2 -13063.16} C_VEL
LIN {X 0,Y 363.736,Z 816.06,A -85,B 0,C 180,E1 -13064.705,E2 -13064.705} C_VEL
LIN {X 0,Y 364.624,Z 806.277,A -85,B 0,C 180,E1 -13065.943,E2 -13065.943} C_VEL
LIN {X 0,Y 365.723,Z 795.285,A -85,B 0,C 180,E1 -13067.042,E2 -13067.042} C_VEL
LIN {X 0,Y 366.797,Z 782.956,A -85,B 0,C 180,E1 -13067.997,E2 -13067.997} C_VEL
LIN {X 0,Y 367.53,Z 771.163,A -85,B 0,C 180,E1 -13068.682,E2 -13068.682} C_VEL
LIN {X 0,Y 368.179,Z 758.245,A -85,B 0,C 180,E1 -13069.189,E2 -13069.189} C_VEL
LIN {X 0,Y 368.671,Z 741.667,A -85,B 0,C 180,E1 -13069.561,E2 -13069.561} C_VEL
LIN {X 0,Y 369.544,Z 675.648,A -85,B 0,C 180,E1 -13070.844,E2 -13070.844} C_VEL
LIN {X 0,Y 365.514,Z 640.557,A -85,B 0,C 180,E1 -13071.805,E2 -13071.805} C_VEL
LIN {X 0,Y 364.913,Z 635.667,A -85,B 0,C 180,E1 -13071.986,E2 -13071.986} C_VEL
LIN {X 0,Y 363.889,Z 623.634,A -85,B 0,C 180,E1 -13072.723,E2 -13072.723} C_VEL
LIN {X 0,Y 365.479,Z 603.888,A -85,B 0,C 180,E1 -13076.557,E2 -13076.557} C_VEL
LIN {X 0,Y 367.311,Z 585.126,A -85,B 0,C 180,E1 -13080.238,E2 -13080.238} C_VEL
LIN {X 0,Y 367.458,Z 580.899,A -85,B 0,C 180,E1 -13081.092,E2 -13081.092} C_VEL
LIN {X 0,Y 364.305,Z 566.067,A -85,B 0,C 180,E1 -13084.352,E2 -13084.352} C_VEL
LIN {X 0,Y 361.874,Z 555.41,A -85,B 0,C 180,E1 -13086.843,E2 -13086.843} C_VEL
LIN {X 0,Y 361.858,Z 555.41,A -85,B 0,C 180,E1 -13089.861,E2 -13089.861} C_VEL
LIN {X 0,Y 361.838,Z 555.413,A -85,B 0,C 180,E1 -13092.829,E2 -13092.829} C_VEL
LIN {X 0,Y 361.838,Z 555.412,A -85,B 0,C 180,E1 -13095.944,E2 -13095.944} C_VEL
LIN {X 0,Y 361.837,Z 555.406,A -85,B 0,C 180,E1 -13099.245,E2 -13099.245} C_VEL
LIN {X 0,Y 361.866,Z 555.4,A -85,B 0,C 180,E1 -13102.777,E2 -13102.777} C_VEL
LIN {X 0,Y 361.856,Z 555.411,A -85,B 0,C 180,E1 -13105.72,E2 -13105.72} C_VEL
LIN {X 0,Y 361.876,Z 555.397,A -85,B 0,C 180,E1 -13109.672,E2 -13109.672} C_VEL
LIN {X 0,Y 361.956,Z 555.392,A -85,B 0,C 180,E1 -13113.475,E2 -13113.475} C_VEL
LIN {X 0,Y 361.883,Z 555.4,A -85,B 0,C 180,E1 -13117.144,E2 -13117.144} C_VEL
LIN {X 0,Y 361.907,Z 555.397,A -85,B 0,C 180,E1 -13120.723,E2 -13120.723} C_VEL
LIN {X 0,Y 361.934,Z 555.383,A -85,B 0,C 180,E1 -13123.066,E2 -13123.066} C_VEL
LIN {X 0,Y 362,Z 555.389,A -85,B 0,C 180,E1 -13126.528,E2 -13126.528} C_VEL
LIN {X 0,Y 362.032,Z 555.369,A -85,B 0,C 180,E1 -13129.938,E2 -13129.938} C_VEL
LIN {X 0,Y 362.163,Z 555.372,A -85,B 0,C 180,E1 -13133.314,E2 -13133.314} C_VEL
LIN {X 0,Y 362.281,Z 555.338,A -85,B 0,C 180,E1 -13137.776,E2 -13137.776} C_VEL
LIN {X 0,Y 362.426,Z 555.339,A -85,B 0,C 180,E1 -13140,E2 -13140} C_VEL
LIN {X 0,Y 362.281,Z 555.354,A -85,B 0,C 180,E1 -13142.224,E2 -13142.224} C_VEL
LIN {X 0,Y 362.163,Z 555.363,A -85,B 0,C 180,E1 -13146.686,E2 -13146.686} C_VEL
LIN {X 0,Y 362.034,Z 555.384,A -85,B 0,C 180,E1 -13150.062,E2 -13150.062} C_VEL
LIN {X 0,Y 361.999,Z 555.382,A -85,B 0,C 180,E1 -13153.899,E2 -13153.899} C_VEL
LIN {X 0,Y 361.969,Z 555.386,A -85,B 0,C 180,E1 -13157.939,E2 -13157.939} C_VEL
LIN {X 0,Y 361.893,Z 555.403,A -85,B 0,C 180,E1 -13161.653,E2 -13161.653} C_VEL
LIN {X 0,Y 361.93,Z 555.387,A -85,B 0,C 180,E1 -13165.29,E2 -13165.29} C_VEL
LIN {X 0,Y 361.91,Z 555.403,A -85,B 0,C 180,E1 -13167.779,E2 -13167.779} C_VEL
LIN {X 0,Y 361.841,Z 555.404,A -85,B 0,C 180,E1 -13171.629,E2 -13171.629} C_VEL
LIN {X 0,Y 361.876,Z 555.401,A -85,B 0,C 180,E1 -13175.345,E2 -13175.345} C_VEL
LIN {X 0,Y 361.871,Z 555.405,A -85,B 0,C 180,E1 -13179.026,E2 -13179.026} C_VEL
LIN {X 0,Y 361.838,Z 555.406,A -85,B 0,C 180,E1 -13182.829,E2 -13182.829} C_VEL
LIN {X 0,Y 361.82,Z 555.407,A -85,B 0,C 180,E1 -13185.947,E2 -13185.947} C_VEL
LIN {X 0,Y 361.838,Z 555.413,A -85,B 0,C 180,E1 -13189.245,E2 -13189.245} C_VEL
LIN {X 0,Y 361.867,Z 555.4,A -85,B 0,C 180,E1 -13192.777,E2 -13192.777} C_VEL
LIN {X 0,Y 361.885,Z 555.498,A -85,B 0,C 180,E1 -13196.091,E2 -13196.091} C_VEL
LIN {X 0,Y 365.79,Z 570.164,A -85,B 0,C 180,E1 -13199.021,E2 -13199.021} C_VEL
LIN {X 0,Y 368.69,Z 583.193,A -85,B 0,C 180,E1 -13201.539,E2 -13201.539} C_VEL
LIN {X 0,Y 368.945,Z 586.74,A -85,B 0,C 180,E1 -13202.179,E2 -13202.179} C_VEL
LIN {X 0,Y 367.362,Z 608.261,A -85,B 0,C 180,E1 -13205.712,E2 -13205.712} C_VEL
LIN {X 0,Y 366.64,Z 623.62,A -85,B 0,C 180,E1 -13208.09,E2 -13208.09} C_VEL
LIN {X 0,Y 370.521,Z 647.76,A -85,B 0,C 180,E1 -13208.835,E2 -13208.835} C_VEL
LIN {X 0,Y 369.269,Z 720.855,A -85,B 0,C 180,E1 -13210.255,E2 -13210.255} C_VEL
LIN {X 0,Y 368.978,Z 737.691,A -85,B 0,C 180,E1 -13210.637,E2 -13210.637} C_VEL
LIN {X 0,Y 368.386,Z 750.61,A -85,B 0,C 180,E1 -13211.147,E2 -13211.147} C_VEL
LIN {X 0,Y 367.569,Z 762.58,A -85,B 0,C 180,E1 -13211.826,E2 -13211.826} C_VEL
LIN {X 0,Y 366.702,Z 774.234,A -85,B 0,C 180,E1 -13212.718,E2 -13212.718} C_VEL
LIN {X 0,Y 365.714,Z 785.052,A -85,B 0,C 180,E1 -13213.782,E2 -13213.782} C_VEL
LIN {X 0,Y 364.781,Z 795.46,A -85,B 0,C 180,E1 -13215.066,E2 -13215.066} C_VEL
LIN {X 0,Y 363.797,Z 803.732,A -85,B 0,C 180,E1 -13216.31,E2 -13216.31} C_VEL
LIN {X 0,Y 362.908,Z 811.36,A -85,B 0,C 180,E1 -13217.7,E2 -13217.7} C_VEL
LIN {X 0,Y 362.063,Z 818.801,A -85,B 0,C 180,E1 -13219.373,E2 -13219.373} C_VEL
LIN {X 0,Y 361.393,Z 824.777,A -85,B 0,C 180,E1 -13221.049,E2 -13221.049} C_VEL
LIN {X 0,Y 360.996,Z 829.499,A -85,B 0,C 180,E1 -13222.729,E2 -13222.729} C_VEL
LIN {X 0,Y 360.714,Z 833.11,A -85,B 0,C 180,E1 -13224.409,E2 -13224.409} C_VEL
LIN {X 0,Y 360.541,Z 834.971,A -85,B 0,C 180,E1 -13225.527,E2 -13225.527} C_VEL
LIN {X 0,Y 360.408,Z 836.393,A -85,B 0,C 180,E1 -13226.645,E2 -13226.645} C_VEL
LIN {X 0,Y 360.35,Z 838.002,A -85,B 0,C 180,E1 -13228.882,E2 -13228.882} C_VEL
LIN {X 0,Y 360.361,Z 838.236,A -85,B 0,C 180,E1 -13229.999,E2 -13229.999} C_VEL
LIN {X 0,Y 360.35,Z 838.045,A -85,B 0,C 180,E1 -13231.117,E2 -13231.117} C_VEL
LIN {X 0,Y 360.399,Z 836.494,A -85,B 0,C 180,E1 -13233.353,E2 -13233.353} C_VEL
LIN {X 0,Y 360.539,Z 835.128,A -85,B 0,C 180,E1 -13234.471,E2 -13234.471} C_VEL
LIN {X 0,Y 360.771,Z 832.171,A -85,B 0,C 180,E1 -13236.191,E2 -13236.191} C_VEL
LIN {X 0,Y 361.061,Z 828.354,A -85,B 0,C 180,E1 -13237.83,E2 -13237.83} C_VEL
LIN {X 0,Y 361.575,Z 823.299,A -85,B 0,C 180,E1 -13239.509,E2 -13239.509} C_VEL
LIN {X 0,Y 362.254,Z 816.927,A -85,B 0,C 180,E1 -13241.186,E2 -13241.186} C_VEL
LIN {X 0,Y 363.183,Z 808.996,A -85,B 0,C 180,E1 -13242.857,E2 -13242.857} C_VEL
LIN {X 0,Y 364.212,Z 800.883,A -85,B 0,C 180,E1 -13244.242,E2 -13244.242} C_VEL
LIN {X 0,Y 365.19,Z 790.926,A -85,B 0,C 180,E1 -13245.629,E2 -13245.629} C_VEL
LIN {X 0,Y 366.228,Z 779.735,A -85,B 0,C 180,E1 -13246.872,E2 -13246.872} C_VEL
LIN {X 0,Y 366.881,Z 772.598,A -85,B 0,C 180,E1 -13247.519,E2 -13247.519} C_VEL
LIN {X 0,Y 366.67,Z 767.428,A -85,B 0,C 180,E1 -13247.962,E2 -13247.962} C_VEL
LIN {X 0,Y 364.602,Z 758.867,A -85,B 0,C 180,E1 -13248.687,E2 -13248.687} C_VEL
LIN {X 0,Y 362.409,Z 750.07,A -85,B 0,C 180,E1 -13249.316,E2 -13249.316} C_VEL
LIN {X 0,Y 361.994,Z 744.468,A -85,B 0,C 180,E1 -13249.6,E2 -13249.6} C_VEL
LIN {X 0,Y 362.499,Z 731.102,A -85,B 0,C 180,E1 -13250.017,E2 -13250.017} C_VEL
LIN {X 0,Y 363.877,Z 651.306,A -85,B 0,C 180,E1 -13251.601,E2 -13251.601} C_VEL
LIN {X 0,Y 359.737,Z 626.912,A -85,B 0,C 180,E1 -13252.381,E2 -13252.381} C_VEL
LIN {X 0,Y 359.308,Z 624.387,A -85,B 0,C 180,E1 -13252.496,E2 -13252.496} C_VEL
LIN {X 0,Y 360.597,Z 603.033,A -85,B 0,C 180,E1 -13256.293,E2 -13256.293} C_VEL
LIN {X 0,Y 361.694,Z 586.678,A -85,B 0,C 180,E1 -13259.38,E2 -13259.38} C_VEL
LIN {X 0,Y 360.744,Z 580.61,A -85,B 0,C 180,E1 -13260.651,E2 -13260.651} C_VEL
LIN {X 0,Y 358.058,Z 568.445,A -85,B 0,C 180,E1 -13263.337,E2 -13263.337} C_VEL
LIN {X 0,Y 354.815,Z 556.284,A -85,B 0,C 180,E1 -13266.082,E2 -13266.082} C_VEL
LIN {X 0,Y 354.82,Z 556.278,A -85,B 0,C 180,E1 -13269.422,E2 -13269.422} C_VEL
LIN {X 0,Y 354.786,Z 556.277,A -85,B 0,C 180,E1 -13272.866,E2 -13272.866} C_VEL
LIN {X 0,Y 354.853,Z 556.282,A -85,B 0,C 180,E1 -13276.117,E2 -13276.117} C_VEL
LIN {X 0,Y 354.89,Z 556.281,A -85,B 0,C 180,E1 -13277.145,E2 -13277.145} C_VEL
LIN {X 0,Y 361.698,Z 575.738,A -85,B 0,C 180,E1 -13277.969,E2 -13277.969} C_VEL
LIN {X 0,Y 360.63,Z 633.867,A -85,B 0,C 180,E1 -13279.329,E2 -13279.329} C_VEL
LIN {X 0,Y 360.522,Z 647.31,A -85,B 0,C 180,E1 -13279.806,E2 -13279.806} C_VEL
LIN {X 0,Y 360.162,Z 661.051,A -85,B 0,C 180,E1 -13280.55,E2 -13280.55} C_VEL
LIN {X 0,Y 359.638,Z 672.919,A -85,B 0,C 180,E1 -13281.412,E2 -13281.412} C_VEL
LIN {X 0,Y 359.034,Z 684.212,A -85,B 0,C 180,E1 -13282.463,E2 -13282.463} C_VEL
LIN {X 0,Y 358.346,Z 695.001,A -85,B 0,C 180,E1 -13283.721,E2 -13283.721} C_VEL
LIN {X 0,Y 357.635,Z 704.564,A -85,B 0,C 180,E1 -13285.086,E2 -13285.086} C_VEL
LIN {X 0,Y 357.01,Z 712.961,A -85,B 0,C 180,E1 -13286.55,E2 -13286.55} C_VEL
LIN {X 0,Y 356.399,Z 720.741,A -85,B 0,C 180,E1 -13288.223,E2 -13288.223} C_VEL
LIN {X 0,Y 355.846,Z 726.805,A -85,B 0,C 180,E1 -13289.825,E2 -13289.825} C_VEL
LIN {X 0,Y 355.523,Z 732.352,A -85,B 0,C 180,E1 -13291.677,E2 -13291.677} C_VEL
LIN {X 0,Y 355.221,Z 736.625,A -85,B 0,C 180,E1 -13293.566,E2 -13293.566} C_VEL
LIN {X 0,Y 355.054,Z 739.731,A -85,B 0,C 180,E1 -13295.575,E2 -13295.575} C_VEL
LIN {X 0,Y 355.024,Z 740.88,A -85,B 0,C 180,E1 -13296.677,E2 -13296.677} C_VEL
LIN {X 0,Y 355.093,Z 741.907,A -85,B 0,C 180,E1 -13298.465,E2 -13298.465} C_VEL
LIN {X 0,Y 355.343,Z 741.872,A -85,B 0,C 180,E1 -13300.353,E2 -13300.353} C_VEL
LIN {X 0,Y 355.543,Z 741.231,A -85,B 0,C 180,E1 -13301.583,E2 -13301.583} C_VEL
LIN {X 0,Y 355.813,Z 740.126,A -85,B 0,C 180,E1 -13302.766,E2 -13302.766} C_VEL
LIN {X 0,Y 356.189,Z 738.553,A -85,B 0,C 180,E1 -13303.964,E2 -13303.964} C_VEL
LIN {X 0,Y 356.801,Z 735.259,A -85,B 0,C 180,E1 -13305.746,E2 -13305.746} C_VEL
LIN {X 0,Y 357.597,Z 730.748,A -85,B 0,C 180,E1 -13307.515,E2 -13307.515} C_VEL
LIN {X 0,Y 358.547,Z 724.76,A -85,B 0,C 180,E1 -13309.311,E2 -13309.311} C_VEL
LIN {X 0,Y 359.568,Z 717.601,A -85,B 0,C 180,E1 -13311.004,E2 -13311.004} C_VEL
LIN {X 0,Y 360.597,Z 709.895,A -85,B 0,C 180,E1 -13312.469,E2 -13312.469} C_VEL
LIN {X 0,Y 361.695,Z 700.277,A -85,B 0,C 180,E1 -13313.94,E2 -13313.94} C_VEL
LIN {X 0,Y 362.812,Z 689.393,A -85,B 0,C 180,E1 -13315.278,E2 -13315.278} C_VEL
LIN {X 0,Y 363.748,Z 677.739,A -85,B 0,C 180,E1 -13316.4,E2 -13316.4} C_VEL
LIN {X 0,Y 364.499,Z 665.568,A -85,B 0,C 180,E1 -13317.306,E2 -13317.306} C_VEL
LIN {X 0,Y 364.913,Z 653.015,A -85,B 0,C 180,E1 -13317.999,E2 -13317.999} C_VEL
LIN {X 0,Y 365.064,Z 639.086,A -85,B 0,C 180,E1 -13318.518,E2 -13318.518} C_VEL
LIN {X 0,Y 365.902,Z 603.726,A -85,B 0,C 180,E1 -13319.424,E2 -13319.424} C_VEL
LIN {X 0,Y 366.628,Z 580.054,A -85,B 0,C 180,E1 -13320.038,E2 -13320.038} C_VEL
LIN {X 0,Y 359.929,Z 565.729,A -85,B 0,C 180,E1 -13321.102,E2 -13321.102} C_VEL
LIN {X 0,Y 355.444,Z 557.411,A -85,B 0,C 180,E1 -13321.82,E2 -13321.82} C_VEL
LIN {X 0,Y 355.189,Z 556.243,A -85,B 0,C 180,E1 -13321.885,E2 -13321.885} C_VEL
LIN {X 0,Y 355.132,Z 556.247,A -85,B 0,C 180,E1 -13326.819,E2 -13326.819} C_VEL
LIN {X 0,Y 355.007,Z 556.263,A -85,B 0,C 180,E1 -13329.113,E2 -13329.113} C_VEL
LIN {X 0,Y 354.916,Z 556.271,A -85,B 0,C 180,E1 -13332.581,E2 -13332.581} C_VEL
LIN {X 0,Y 354.88,Z 556.272,A -85,B 0,C 180,E1 -13336.096,E2 -13336.096} C_VEL
LIN {X 0,Y 354.896,Z 556.278,A -85,B 0,C 180,E1 -13338.472,E2 -13338.472} C_VEL
LIN {X 0,Y 354.825,Z 556.286,A -85,B 0,C 180,E1 -13342.107,E2 -13342.107} C_VEL
LIN {X 0,Y 354.89,Z 556.276,A -85,B 0,C 180,E1 -13345.828,E2 -13345.828} C_VEL
LIN {X 0,Y 354.846,Z 556.283,A -85,B 0,C 180,E1 -13349.679,E2 -13349.679} C_VEL
LIN {X 0,Y 354.798,Z 556.289,A -85,B 0,C 180,E1 -13353.703,E2 -13353.703} C_VEL
LIN {X 0,Y 354.792,Z 556.293,A -85,B 0,C 180,E1 -13356.46,E2 -13356.46} C_VEL
LIN {X 0,Y 354.817,Z 556.287,A -85,B 0,C 180,E1 -13359.425,E2 -13359.425} C_VEL
LIN {X 0,Y 354.835,Z 556.284,A -85,B 0,C 180,E1 -13362.878,E2 -13362.878} C_VEL
LIN {X 0,Y 354.862,Z 556.285,A -85,B 0,C 180,E1 -13366.121,E2 -13366.121} C_VEL
LIN {X 0,Y 354.851,Z 556.282,A -85,B 0,C 180,E1 -13369.19,E2 -13369.19} C_VEL
LIN {X 0,Y 354.845,Z 556.404,A -85,B 0,C 180,E1 -13372.034,E2 -13372.034} C_VEL
LIN {X 0,Y 358.17,Z 567.977,A -85,B 0,C 180,E1 -13375.319,E2 -13375.319} C_VEL
LIN {X 0,Y 360.986,Z 579.853,A -85,B 0,C 180,E1 -13378.289,E2 -13378.289} C_VEL
LIN {X 0,Y 362.17,Z 586.047,A -85,B 0,C 180,E1 -13379.701,E2 -13379.701} C_VEL
LIN {X 0,Y 360.99,Z 595.656,A -85,B 0,C 180,E1 -13381.586,E2 -13381.586} C_VEL
LIN {X 0,Y 358.807,Z 614.244,A -85,B 0,C 180,E1 -13385.096,E2 -13385.096} C_VEL
LIN {X 0,Y 358.318,Z 619.438,A -85,B 0,C 180,E1 -13386.024,E2 -13386.024} C_VEL
LIN {X 0,Y 361.859,Z 642.933,A -85,B 0,C 180,E1 -13387.017,E2 -13387.017} C_VEL
LIN {X 0,Y 364.006,Z 666.148,A -85,B 0,C 180,E1 -13387.842,E2 -13387.842} C_VEL
LIN {X 0,Y 364.557,Z 677.869,A -85,B 0,C 180,E1 -13388.209,E2 -13388.209} C_VEL
LIN {X 0,Y 362.762,Z 733.9,A -85,B 0,C 180,E1 -13389.592,E2 -13389.592} C_VEL
LIN {X 0,Y 361.92,Z 747.284,A -85,B 0,C 180,E1 -13390.135,E2 -13390.135} C_VEL
LIN {X 0,Y 361.262,Z 763.389,A -85,B 0,C 180,E1 -13390.615,E2 -13390.615} C_VEL
LIN {X 0,Y 360.45,Z 776.401,A -85,B 0,C 180,E1 -13391.235,E2 -13391.235} C_VEL
LIN {X 0,Y 359.53,Z 788.643,A -85,B 0,C 180,E1 -13392.07,E2 -13392.07} C_VEL
LIN {X 0,Y 358.537,Z 799.641,A -85,B 0,C 180,E1 -13393.049,E2 -13393.049} C_VEL
LIN {X 0,Y 357.431,Z 810.382,A -85,B 0,C 180,E1 -13394.255,E2 -13394.255} C_VEL
LIN {X 0,Y 356.312,Z 820.733,A -85,B 0,C 180,E1 -13395.728,E2 -13395.728} C_VEL
LIN {X 0,Y 355.467,Z 828.841,A -85,B 0,C 180,E1 -13397.15,E2 -13397.15} C_VEL
LIN {X 0,Y 354.59,Z 836.774,A -85,B 0,C 180,E1 -13398.859,E2 -13398.859} C_VEL
LIN {X 0,Y 354.078,Z 842.128,A -85,B 0,C 180,E1 -13400.288,E2 -13400.288} C_VEL
LIN {X 0,Y 353.683,Z 847.357,A -85,B 0,C 180,E1 -13402.006,E2 -13402.006} C_VEL
LIN {X 0,Y 353.439,Z 851.641,A -85,B 0,C 180,E1 -13403.844,E2 -13403.844} C_VEL
LIN {X 0,Y 353.376,Z 854.377,A -85,B 0,C 180,E1 -13405.438,E2 -13405.438} C_VEL
LIN {X 0,Y 353.304,Z 855.805,A -85,B 0,C 180,E1 -13406.58,E2 -13406.58} C_VEL
LIN {X 0,Y 353.349,Z 857.429,A -85,B 0,C 180,E1 -13408.861,E2 -13408.861} C_VEL
LIN {X 0,Y 353.409,Z 857.649,A -85,B 0,C 180,E1 -13410.001,E2 -13410.001} C_VEL
LIN {X 0,Y 353.328,Z 857.423,A -85,B 0,C 180,E1 -13411.141,E2 -13411.141} C_VEL
LIN {X 0,Y 353.294,Z 855.791,A -85,B 0,C 180,E1 -13413.422,E2 -13413.422} C_VEL
LIN {X 0,Y 353.366,Z 854.357,A -85,B 0,C 180,E1 -13414.564,E2 -13414.564} C_VEL
LIN {X 0,Y 353.39,Z 851.76,A -85,B 0,C 180,E1 -13416.082,E2 -13416.082} C_VEL
LIN {X 0,Y 353.683,Z 847.322,A -85,B 0,C 180,E1 -13417.996,E2 -13417.996} C_VEL
LIN {X 0,Y 354.168,Z 841.072,A -85,B 0,C 180,E1 -13420,E2 -13420} C_VEL
LIN {X 0,Y 354.801,Z 834.254,A -85,B 0,C 180,E1 -13421.715,E2 -13421.715} C_VEL
LIN {X 0,Y 355.792,Z 825.723,A -85,B 0,C 180,E1 -13423.421,E2 -13423.421} C_VEL
LIN {X 0,Y 356.738,Z 816.934,A -85,B 0,C 180,E1 -13424.84,E2 -13424.84} C_VEL
LIN {X 0,Y 357.671,Z 807.267,A -85,B 0,C 180,E1 -13426.115,E2 -13426.115} C_VEL
LIN {X 0,Y 358.8,Z 796.663,A -85,B 0,C 180,E1 -13427.234,E2 -13427.234} C_VEL
LIN {X 0,Y 359.86,Z 784.747,A -85,B 0,C 180,E1 -13428.209,E2 -13428.209} C_VEL
LIN {X 0,Y 360.699,Z 772.329,A -85,B 0,C 180,E1 -13428.975,E2 -13428.975} C_VEL
LIN {X 0,Y 361.423,Z 760.312,A -85,B 0,C 180,E1 -13429.489,E2 -13429.489} C_VEL
LIN {X 0,Y 361.897,Z 746.965,A -85,B 0,C 180,E1 -13429.831,E2 -13429.831} C_VEL
LIN {X 0,Y 362.868,Z 675.919,A -85,B 0,C 180,E1 -13431.238,E2 -13431.238} C_VEL
LIN {X 0,Y 358.984,Z 641.886,A -85,B 0,C 180,E1 -13432.193,E2 -13432.193} C_VEL
LIN {X 0,Y 358.171,Z 635.516,A -85,B 0,C 180,E1 -13432.422,E2 -13432.422} C_VEL
LIN {X 0,Y 357.065,Z 621.529,A -85,B 0,C 180,E1 -13433.336,E2 -13433.336} C_VEL
LIN {X 0,Y 358.855,Z 601.048,A -85,B 0,C 180,E1 -13437.403,E2 -13437.403} C_VEL
LIN {X 0,Y 360.595,Z 583.369,A -85,B 0,C 180,E1 -13440.956,E2 -13440.956} C_VEL
LIN {X 0,Y 358.899,Z 574.522,A -85,B 0,C 180,E1 -13442.901,E2 -13442.901} C_VEL
LIN {X 0,Y 355.586,Z 559.478,A -85,B 0,C 180,E1 -13446.366,E2 -13446.366} C_VEL
LIN {X 0,Y 354.826,Z 556.288,A -85,B 0,C 180,E1 -13447.165,E2 -13447.165} C_VEL
LIN {X 0,Y 354.79,Z 556.292,A -85,B 0,C 180,E1 -13450.821,E2 -13450.821} C_VEL
LIN {X 0,Y 354.791,Z 556.28,A -85,B 0,C 180,E1 -13454.511,E2 -13454.511} C_VEL
LIN {X 0,Y 354.796,Z 556.28,A -85,B 0,C 180,E1 -13457.663,E2 -13457.663} C_VEL
LIN {X 0,Y 354.817,Z 556.287,A -85,B 0,C 180,E1 -13460.666,E2 -13460.666} C_VEL
LIN {X 0,Y 354.824,Z 556.278,A -85,B 0,C 180,E1 -13464.301,E2 -13464.301} C_VEL
LIN {X 0,Y 354.788,Z 556.282,A -85,B 0,C 180,E1 -13467.667,E2 -13467.667} C_VEL
LIN {X 0,Y 354.87,Z 556.274,A -85,B 0,C 180,E1 -13470.621,E2 -13470.621} C_VEL
LIN {X 0,Y 354.9,Z 556.265,A -85,B 0,C 180,E1 -13474.173,E2 -13474.173} C_VEL
LIN {X 0,Y 354.818,Z 556.287,A -85,B 0,C 180,E1 -13477.893,E2 -13477.893} C_VEL
LIN {X 0,Y 354.923,Z 556.253,A -85,B 0,C 180,E1 -13481.892,E2 -13481.892} C_VEL
LIN {X 0,Y 354.944,Z 556.27,A -85,B 0,C 180,E1 -13485.981,E2 -13485.981} C_VEL
LIN {X 0,Y 354.979,Z 556.246,A -85,B 0,C 180,E1 -13489.736,E2 -13489.736} C_VEL
LIN {X 0,Y 355.127,Z 556.248,A -85,B 0,C 180,E1 -13493.181,E2 -13493.181} C_VEL
LIN {X 0,Y 355.244,Z 556.213,A -85,B 0,C 180,E1 -13497.732,E2 -13497.732} C_VEL
LIN {X 0,Y 355.375,Z 556.217,A -85,B 0,C 180,E1 -13500,E2 -13500} C_VEL
LIN {X 0,Y 355.244,Z 556.23,A -85,B 0,C 180,E1 -13502.268,E2 -13502.268} C_VEL
LIN {X 0,Y 355.128,Z 556.24,A -85,B 0,C 180,E1 -13506.819,E2 -13506.819} C_VEL
LIN {X 0,Y 354.98,Z 556.26,A -85,B 0,C 180,E1 -13510.264,E2 -13510.264} C_VEL
LIN {X 0,Y 354.944,Z 556.262,A -85,B 0,C 180,E1 -13514.019,E2 -13514.019} C_VEL
LIN {X 0,Y 354.924,Z 556.261,A -85,B 0,C 180,E1 -13518.108,E2 -13518.108} C_VEL
LIN {X 0,Y 354.836,Z 556.288,A -85,B 0,C 180,E1 -13522.106,E2 -13522.106} C_VEL
LIN {X 0,Y 354.9,Z 556.263,A -85,B 0,C 180,E1 -13525.827,E2 -13525.827} C_VEL
LIN {X 0,Y 354.819,Z 556.283,A -85,B 0,C 180,E1 -13529.682,E2 -13529.682} C_VEL
LIN {X 0,Y 354.833,Z 556.288,A -85,B 0,C 180,E1 -13533.682,E2 -13533.682} C_VEL
LIN {X 0,Y 354.8,Z 556.288,A -85,B 0,C 180,E1 -13536.459,E2 -13536.459} C_VEL
LIN {X 0,Y 354.826,Z 556.282,A -85,B 0,C 180,E1 -13539.424,E2 -13539.424} C_VEL
LIN {X 0,Y 354.79,Z 556.284,A -85,B 0,C 180,E1 -13542.867,E2 -13542.867} C_VEL
LIN {X 0,Y 354.769,Z 556.282,A -85,B 0,C 180,E1 -13546.103,E2 -13546.103} C_VEL
LIN {X 0,Y 354.79,Z 556.289,A -85,B 0,C 180,E1 -13549.179,E2 -13549.179} C_VEL
LIN {X 0,Y 354.81,Z 556.276,A -85,B 0,C 180,E1 -13552.402,E2 -13552.402} C_VEL
LIN {X 0,Y 354.841,Z 556.345,A -85,B 0,C 180,E1 -13555.591,E2 -13555.591} C_VEL
LIN {X 0,Y 358.548,Z 569.998,A -85,B 0,C 180,E1 -13558.376,E2 -13558.376} C_VEL
LIN {X 0,Y 361.591,Z 583.342,A -85,B 0,C 180,E1 -13561.002,E2 -13561.002} C_VEL
LIN {X 0,Y 362.234,Z 586.727,A -85,B 0,C 180,E1 -13561.653,E2 -13561.653} C_VEL
LIN {X 0,Y 360.981,Z 604.646,A -85,B 0,C 180,E1 -13564.638,E2 -13564.638} C_VEL
LIN {X 0,Y 359.918,Z 623.754,A -85,B 0,C 180,E1 -13567.66,E2 -13567.66} C_VEL
LIN {X 0,Y 363.885,Z 648.829,A -85,B 0,C 180,E1 -13568.451,E2 -13568.451} C_VEL
LIN {X 0,Y 362.401,Z 735.385,A -85,B 0,C 180,E1 -13570.197,E2 -13570.197} C_VEL
LIN {X 0,Y 361.756,Z 748.653,A -85,B 0,C 180,E1 -13570.678,E2 -13570.678} C_VEL
LIN {X 0,Y 361.061,Z 760.615,A -85,B 0,C 180,E1 -13571.339,E2 -13571.339} C_VEL
LIN {X 0,Y 360.115,Z 772.799,A -85,B 0,C 180,E1 -13572.245,E2 -13572.245} C_VEL
LIN {X 0,Y 359.096,Z 783.312,A -85,B 0,C 180,E1 -13573.25,E2 -13573.25} C_VEL
LIN {X 0,Y 358.144,Z 793.576,A -85,B 0,C 180,E1 -13574.492,E2 -13574.492} C_VEL
LIN {X 0,Y 356.909,Z 803.922,A -85,B 0,C 180,E1 -13576.041,E2 -13576.041} C_VEL
LIN {X 0,Y 355.823,Z 812.884,A -85,B 0,C 180,E1 -13577.74,E2 -13577.74} C_VEL
LIN {X 0,Y 354.957,Z 820.082,A -85,B 0,C 180,E1 -13579.446,E2 -13579.446} C_VEL
LIN {X 0,Y 354.2,Z 826.691,A -85,B 0,C 180,E1 -13581.441,E2 -13581.441} C_VEL
LIN {X 0,Y 353.794,Z 831.402,A -85,B 0,C 180,E1 -13583.333,E2 -13583.333} C_VEL
LIN {X 0,Y 353.481,Z 835.163,A -85,B 0,C 180,E1 -13585.438,E2 -13585.438} C_VEL
LIN {X 0,Y 353.329,Z 836.586,A -85,B 0,C 180,E1 -13586.578,E2 -13586.578} C_VEL
LIN {X 0,Y 353.253,Z 838.195,A -85,B 0,C 180,E1 -13588.859,E2 -13588.859} C_VEL
LIN {X 0,Y 353.264,Z 838.429,A -85,B 0,C 180,E1 -13589.999,E2 -13589.999} C_VEL
LIN {X 0,Y 353.252,Z 838.238,A -85,B 0,C 180,E1 -13591.139,E2 -13591.139} C_VEL
LIN {X 0,Y 353.321,Z 836.686,A -85,B 0,C 180,E1 -13593.42,E2 -13593.42} C_VEL
LIN {X 0,Y 353.478,Z 835.319,A -85,B 0,C 180,E1 -13594.561,E2 -13594.561} C_VEL
LIN {X 0,Y 353.784,Z 831.646,A -85,B 0,C 180,E1 -13596.653,E2 -13596.653} C_VEL
LIN {X 0,Y 354.193,Z 826.973,A -85,B 0,C 180,E1 -13598.557,E2 -13598.557} C_VEL
LIN {X 0,Y 354.829,Z 821.52,A -85,B 0,C 180,E1 -13600.267,E2 -13600.267} C_VEL
LIN {X 0,Y 355.628,Z 814.681,A -85,B 0,C 180,E1 -13601.975,E2 -13601.975} C_VEL
LIN {X 0,Y 356.655,Z 806.109,A -85,B 0,C 180,E1 -13603.677,E2 -13603.677} C_VEL
LIN {X 0,Y 357.745,Z 797.338,A -85,B 0,C 180,E1 -13605.085,E2 -13605.085} C_VEL
LIN {X 0,Y 358.778,Z 786.944,A -85,B 0,C 180,E1 -13606.441,E2 -13606.441} C_VEL
LIN {X 0,Y 359.862,Z 775.493,A -85,B 0,C 180,E1 -13607.619,E2 -13607.619} C_VEL
LIN {X 0,Y 360.749,Z 765.153,A -85,B 0,C 180,E1 -13608.455,E2 -13608.455} C_VEL
LIN {X 0,Y 361.648,Z 752.771,A -85,B 0,C 180,E1 -13609.216,E2 -13609.216} C_VEL
LIN {X 0,Y 361.994,Z 744.468,A -85,B 0,C 180,E1 -13609.6,E2 -13609.6} C_VEL
LIN {X 0,Y 361.563,Z 738.774,A -85,B 0,C 180,E1 -13609.848,E2 -13609.848} C_VEL
LIN {X 0,Y 356.726,Z 721.121,A -85,B 0,C 180,E1 -13610.577,E2 -13610.577} C_VEL
LIN {X 0,Y 356.169,Z 716.303,A -85,B 0,C 180,E1 -13610.708,E2 -13610.708} C_VEL
LIN {X 0,Y 356.196,Z 714.351,A -85,B 0,C 180,E1 -13610.747,E2 -13610.747} C_VEL
LIN {X 0,Y 357.235,Z 651.355,A -85,B 0,C 180,E1 -13612.023,E2 -13612.023} C_VEL
LIN {X 0,Y 352.715,Z 625.568,A -85,B 0,C 180,E1 -13612.881,E2 -13612.881} C_VEL
LIN {X 0,Y 352.587,Z 624.272,A -85,B 0,C 180,E1 -13612.996,E2 -13612.996} C_VEL
LIN {X 0,Y 353.873,Z 603.854,A -85,B 0,C 180,E1 -13616.656,E2 -13616.656} C_VEL
LIN {X 0,Y 354.925,Z 588.066,A -85,B 0,C 180,E1 -13619.67,E2 -13619.67} C_VEL
LIN {X 0,Y 353.117,Z 578.096,A -85,B 0,C 180,E1 -13621.829,E2 -13621.829} C_VEL
LIN {X 0,Y 350.141,Z 565.814,A -85,B 0,C 180,E1 -13624.619,E2 -13624.619} C_VEL
LIN {X 0,Y 347.767,Z 557.164,A -85,B 0,C 180,E1 -13626.641,E2 -13626.641} C_VEL
LIN {X 0,Y 347.729,Z 557.165,A -85,B 0,C 180,E1 -13630.295,E2 -13630.295} C_VEL
LIN {X 0,Y 347.723,Z 557.153,A -85,B 0,C 180,E1 -13633.406,E2 -13633.406} C_VEL
LIN {X 0,Y 347.816,Z 557.162,A -85,B 0,C 180,E1 -13636.826,E2 -13636.826} C_VEL
